(* IEC 61131-3 sources: Industry-PLC-LLM/data/PLCBEAD_repo/PLCBEAD_PLCEmbed-main/PLC-BEAD/Source/OpenPLCv2 (part 4) *)

(* ---- DIR_TO_DEG.ST ---- *)
TYPE oscat_LANGUAGE:
  STRUCT
    DEFAULT 	: INT;
	LMAX    	: INT;
  END_STRUCT;
END_TYPE

TYPE
  oscat_ELEMENT_DIRS 		: ARRAY [0..15] OF STRING;
  oscat_DIRS				: ARRAY [1..3]  OF oscat_ELEMENT_DIRS := [0,0 , 0];
END_TYPE

FUNCTION_BLOCK SETUP_DIRS
	VAR_IN_OUT
		DIRS :	oscat_DIRS;
	END_VAR

	VAR
		init :	BOOL;
	END_VAR

	IF init THEN RETURN; END_IF;
	init := TRUE;

	(* ---- english --- *)
	DIRS[1][00] := 'N';
	DIRS[1][01] := 'NNE';
	DIRS[1][02] := 'NE';
	DIRS[1][03] := 'ENE';
	DIRS[1][04] := 'E';
	DIRS[1][05] := 'ESE';
	DIRS[1][06] := 'SE';
	DIRS[1][07] := 'SSE';
	DIRS[1][08] := 'S';
	DIRS[1][09] := 'SSW';
	DIRS[1][10] := 'SW';
	DIRS[1][11] := 'WSW';
	DIRS[1][12] := 'W';
	DIRS[1][13] := 'WNW';
	DIRS[1][14] := 'NW';
	DIRS[1][15] := 'NNW';

	(* ---- german --- *)
	DIRS[2][00] := 'N';
	DIRS[2][01] := 'NNO';
	DIRS[2][02] := 'NO';
	DIRS[2][03] := 'ONO';
	DIRS[2][04] := 'O';
	DIRS[2][05] := 'OSO';
	DIRS[2][06] := 'SO';
	DIRS[2][07] := 'SSO';
	DIRS[2][08] := 'S';
	DIRS[2][09] := 'SSW';
	DIRS[2][10] := 'SW';
	DIRS[2][11] := 'WSW';
	DIRS[2][12] := 'W';
	DIRS[2][13] := 'WNW';
	DIRS[2][14] := 'NW';
	DIRS[2][15] := 'NNW';

	(* ---- french --- *)
	DIRS[3][00] := 'N';
	DIRS[3][01] := 'NNO';
	DIRS[3][02] := 'NO';
	DIRS[3][03] := 'ONO';
	DIRS[3][04] := 'O';
	DIRS[3][05] := 'OSO';
	DIRS[3][06] := 'SO';
	DIRS[3][07] := 'SSO';
	DIRS[3][08] := 'S';
	DIRS[3][09] := 'SSW';
	DIRS[3][10] := 'SW';
	DIRS[3][11] := 'WSW';
	DIRS[3][12] := 'W';
	DIRS[3][13] := 'WNW';
	DIRS[3][14] := 'NW';
	DIRS[3][15] := 'NNW';
END_FUNCTION_BLOCK

FUNCTION_BLOCK SETUP_LANGUAGE_Block

	VAR_IN_OUT
		LANGUAGE :	oscat_LANGUAGE;
	END_VAR

	VAR
		init :	BOOL;
	END_VAR

	IF init THEN RETURN; END_IF;
	init := TRUE;

	LANGUAGE.DEFAULT  := 1; (* 1=english, 2=german 3=french *)
	LANGUAGE.LMAX := 3;

END_FUNCTION_BLOCK

FUNCTION_BLOCK DIR_TO_DEG_Block
	VAR_INPUT
		DIR :	STRING;
		L :	INT;
	END_VAR

	VAR_OUTPUT
		DIR_TO_DEG :	INT;
	END_VAR

	VAR
		ly :	INT;
		i :	INT;
		SETUP_DIRSS :	SETUP_DIRS;
		DIRS :	oscat_DIRS;
		SETUP_LANGUAGE :	SETUP_LANGUAGE_Block;
		LANGUAGE :	oscat_LANGUAGE;
	END_VAR

	SETUP_DIRSS(DIRS:=DIRS);
	DIRS:=SETUP_DIRSS.DIRS;
	SETUP_LANGUAGE(LANGUAGE:=LANGUAGE);
	LANGUAGE:=SETUP_LANGUAGE.LANGUAGE;

	IF L = 0 THEN ly := LANGUAGE.DEFAULT; ELSE ly := MIN(L, LANGUAGE.LMAX); END_IF;
	FOR i := 0 TO 15 DO
		IF EQ_STRING(DIRS[ly][i],DIR) THEN EXIT; END_IF;
	END_FOR;
	DIR_TO_DEG := WORD_TO_INT(SHR(INT_TO_WORD(i * 45 + 1), 1));

END_FUNCTION_BLOCK

PROGRAM program0
  VAR
    LocalVar0 : STRING;
	LocalVar1 : INT;

	LocalOUT  : INT;
	func_block : DIR_TO_DEG_Block;
  END_VAR
	func_block.DIR  := LocalVar0;
	func_block.L  := LocalVar1;
	func_block();
	LocalOUT := func_block.DIR_TO_DEG;
END_PROGRAM

CONFIGURATION Config0
  RESOURCE Res0 ON PLC
    TASK task0(INTERVAL := T#20ms,PRIORITY := 0);
    PROGRAM instance0 WITH task0 : program0;
  END_RESOURCE
END_CONFIGURATION

(* ---- DRIVER_1.ST ---- *)
FUNCTION_BLOCK DRIVER_1
	VAR_INPUT
		SET :	BOOL;
		IN :	BOOL;
		RST :	BOOL;
		TOGGLE_MODE :	BOOL;
		TIMEOUT :	TIME;
	END_VAR

	VAR_OUTPUT
		Q :	BOOL;
	END_VAR

	VAR
		off :	TON;
		edge :	BOOL;
	END_VAR

	IF off.Q THEN Q := FALSE; END_IF;
	IF rst THEN
		Q := FALSE;
	ELSIF set THEN
		Q := TRUE;
	ELSIF IN AND NOT edge THEN
		IF toggle_mode THEN q := NOT Q; ELSE q := TRUE; END_IF;
	END_IF;
	edge := in;
	IF timeout > t#0s THEN off(in := Q, PT := Timeout); END_IF;

END_FUNCTION_BLOCK

PROGRAM program0
  VAR
	SET         :	BOOL;
	IN          :	BOOL;
	RST         :	BOOL;
	TOGGLE_MODE :	BOOL;
	TIMEOUT     :	TIME;

	Q :	BOOL;

	func_block : DRIVER_1;
  END_VAR
	func_block.SET         :=SET        ;
	func_block.IN          :=IN         ;
	func_block.RST         :=RST        ;
	func_block.TOGGLE_MODE :=TOGGLE_MODE;
	func_block.TIMEOUT     :=TIMEOUT    ;
	func_block();
	Q := func_block.Q;
END_PROGRAM

CONFIGURATION Config0
  RESOURCE Res0 ON PLC
    TASK task0(INTERVAL := T#20ms,PRIORITY := 0);
    PROGRAM instance0 WITH task0 : program0;
  END_RESOURCE
END_CONFIGURATION

(* ---- DRIVER_4.ST ---- *)
FUNCTION_BLOCK DRIVER_1
	VAR_INPUT
		SET :	BOOL;
		IN :	BOOL;
		RST :	BOOL;
		TOGGLE_MODE :	BOOL;
		TIMEOUT :	TIME;
	END_VAR

	VAR_OUTPUT
		Q :	BOOL;
	END_VAR

	VAR
		off :	TON;
		edge :	BOOL;
	END_VAR

	IF off.Q THEN Q := FALSE; END_IF;
	IF rst THEN
		Q := FALSE;
	ELSIF set THEN
		Q := TRUE;
	ELSIF IN AND NOT edge THEN
		IF toggle_mode THEN q := NOT Q; ELSE q := TRUE; END_IF;
	END_IF;
	edge := in;
	IF timeout > t#0s THEN off(in := Q, PT := Timeout); END_IF;

END_FUNCTION_BLOCK

FUNCTION_BLOCK DRIVER_4

	VAR_INPUT
		SET :	BOOL;
		IN0 :	BOOL;
		IN1 :	BOOL;
		IN2 :	BOOL;
		IN3 :	BOOL;
		RST :	BOOL;
		TOGGLE_MODE :	BOOL;
		TIMEOUT :	TIME;
	END_VAR

	VAR_OUTPUT
		Q0 :	BOOL;
		Q1 :	BOOL;
		Q2 :	BOOL;
		Q3 :	BOOL;
	END_VAR

	VAR
		d0 :	DRIVER_1;
		d1 :	DRIVER_1;
		d2 :	DRIVER_1;
		d3 :	DRIVER_1;
	END_VAR

	D0(Set:=set, in:=in0, rst:=rst, toggle_mode:=toggle_mode, timeout:=timeout);
	D1(Set:=set, in:=in1, rst:=rst, toggle_mode:=toggle_mode, timeout:=timeout);
	D2(Set:=set, in:=in2, rst:=rst, toggle_mode:=toggle_mode, timeout:=timeout);
	D3(Set:=set, in:=in3, rst:=rst, toggle_mode:=toggle_mode, timeout:=timeout);
	Q0 := D0.Q;
	Q1 := D1.Q;
	Q2 := D2.Q;
	Q3 := D3.Q;

END_FUNCTION_BLOCK

PROGRAM program0
  VAR
	SET         :	BOOL;
	IN0         :	BOOL;
	IN1         :	BOOL;
	IN2         :	BOOL;
	IN3         :	BOOL;
	RST         :	BOOL;
	TOGGLE_MODE :	BOOL;
	TIMEOUT     :	TIME;

	Q0 :	BOOL;
	Q1 :	BOOL;
	Q2 :	BOOL;
	Q3 :	BOOL;

	func_block : DRIVER_4;
  END_VAR
	func_block.SET         := SET        ;
	func_block.IN0         := IN0        ;
	func_block.IN1         := IN1        ;
	func_block.IN2         := IN2        ;
	func_block.IN3         := IN3        ;
	func_block.RST         := RST        ;
	func_block.TOGGLE_MODE := TOGGLE_MODE;
	func_block.TIMEOUT     := TIMEOUT    ;
	func_block();
	Q0 := func_block.Q0;
	Q1 := func_block.Q1;
	Q2 := func_block.Q2;
	Q3 := func_block.Q3;
END_PROGRAM

CONFIGURATION Config0
  RESOURCE Res0 ON PLC
    TASK task0(INTERVAL := T#20ms,PRIORITY := 0);
    PROGRAM instance0 WITH task0 : program0;
  END_RESOURCE
END_CONFIGURATION

(* ---- DRIVER_4C.ST ---- *)
TYPE
  oscat_DRIVER_4C 			  : ARRAY [1..7] 	OF BYTE;
END_TYPE
FUNCTION_BLOCK DRIVER_4C

	VAR_INPUT
		IN :	BOOL;
		RST :	BOOL;
		TIMEOUT :	TIME;
		SX :	oscat_DRIVER_4C;
	END_VAR

	VAR_OUTPUT
		SN :	INT;
		Q0 :	BOOL;
		Q1 :	BOOL;
		Q2 :	BOOL;
		Q3 :	BOOL;
	END_VAR

	VAR
		off :	TON;
		edge :	BOOL;
	END_VAR

	IF RST OR off.Q THEN
		SN := 0;
	ELSIF IN AND NOT edge THEN
		SN := SN + 1;
		IF SN > 7 OR SX[SN] = BYTE#0 THEN SN := 0; END_IF;
	END_IF;
	edge := in;
	IF SN > 0 THEN
		Q0 := (SX[SN] AND BYTE#1) > BYTE#0;
		Q1 := (SX[SN] AND BYTE#2) > BYTE#0;
		Q2 := (SX[SN] AND BYTE#4) > BYTE#0;
		Q3 := (SX[SN] AND BYTE#8) > BYTE#0;
	ELSE
		Q0 := FALSE;
		Q1 := FALSE;
		Q2 := FALSE;
		Q3 := FALSE;
	END_IF;

	IF timeout > t#0s THEN off(in := SN > 0, PT := Timeout); END_IF;

END_FUNCTION_BLOCK

PROGRAM program0
  VAR
	IN      :	BOOL;
	RST     :	BOOL;
	TIMEOUT :	TIME;
	SX      :	oscat_DRIVER_4C;

	SN :	INT;
	Q0 :	BOOL;
	Q1 :	BOOL;
	Q2 :	BOOL;
	Q3 :	BOOL;

	func_block : DRIVER_4C;
  END_VAR
	func_block.IN       :=IN      ;
	func_block.RST      :=RST     ;
	func_block.TIMEOUT  :=TIMEOUT ;
	func_block.SX       :=SX      ;
	func_block();
	SN := func_block.SN;
	Q0 := func_block.Q0;
	Q1 := func_block.Q1;
	Q2 := func_block.Q2;
	Q3 := func_block.Q3;
END_PROGRAM

CONFIGURATION Config0
  RESOURCE Res0 ON PLC
    TASK task0(INTERVAL := T#20ms,PRIORITY := 0);
    PROGRAM instance0 WITH task0 : program0;
  END_RESOURCE
END_CONFIGURATION

(* ---- DT2_TO_SDT.ST ---- *)
TYPE oscat_SDT :
STRUCT
	YEAR : INT;
	MONTH : INT;
	DAY : INT;
	WEEKDAY : INT;
	HOUR : INT;
	MINUTE : INT;
	SECOND : INT;
	MS : INT;
END_STRUCT;
END_TYPE

FUNCTION DAY_OF_WEEK:INT

	VAR_INPUT
		IDATE :	UDINT;
	END_VAR

	DAY_OF_WEEK := UDINT_TO_INT((idate / UDINT#86400 + UDINT#3) MOD UDINT#7) + INT#01;
END_FUNCTION

FUNCTION DAY_OF_YEAR:INT
	VAR_INPUT
		IDATE :	UDINT;
	END_VAR

	DAY_OF_YEAR := UDINT_TO_INT(((idate) / UDINT#86400) MOD UDINT#1461);
	IF DAY_OF_YEAR > 729 THEN
		IF DAY_OF_YEAR > 1095 THEN DAY_OF_YEAR := DAY_OF_YEAR - 1095; ELSE DAY_OF_YEAR := DAY_OF_YEAR - 729; END_IF;
	ELSIF DAY_OF_YEAR > 364 THEN
		DAY_OF_YEAR := DAY_OF_YEAR - 364;
	ELSE
		DAY_OF_YEAR := DAY_OF_YEAR + 1;
	END_IF;
END_FUNCTION

FUNCTION LEAP_OF_DATE:BOOL

	VAR_INPUT
		IDATE :	UDINT;
	END_VAR

	LEAP_OF_DATE := SHL(UDINT_TO_DWORD((idate + UDINT#43200) / UDINT#31557600), 30) = DWORD#16#80000000;
END_FUNCTION

FUNCTION DAY_OF_MONTH:INT
	VAR_INPUT
		IDATE :	UDINT;
	END_VAR

	day_of_month := day_of_year(idate);

	IF leap_of_Date(idate) THEN
		CASE day_of_month OF
			32..60	:	day_of_month := day_of_month - 31;
			61..91	:	day_of_month := day_of_month - 60;
			92..121 :	day_of_month := day_of_month - 91;
			122..152:	day_of_month := day_of_month - 121;
			153..182:	day_of_month := day_of_month - 152;
			183..213:	day_of_month := day_of_month - 182;
			214..244:	day_of_month := day_of_month - 213;
			245..274:	day_of_month := day_of_month - 244;
			275..305:	day_of_month := day_of_month - 274;
			306..335:	day_of_month := day_of_month - 305;
			336..366:	day_of_month := day_of_month - 335;
		END_CASE;
	ELSE
		CASE day_of_month OF
			32..59	:	day_of_month := day_of_month - 31;
			60..90	:	day_of_month := day_of_month - 59;
			91..120 :	day_of_month := day_of_month - 90;
			121..151:	day_of_month := day_of_month - 120;
			152..181:	day_of_month := day_of_month - 151;
			182..212:	day_of_month := day_of_month - 181;
			213..243:	day_of_month := day_of_month - 212;
			244..273:	day_of_month := day_of_month - 243;
			274..304:	day_of_month := day_of_month - 273;
			305..334:	day_of_month := day_of_month - 304;
			335..365:	day_of_month := day_of_month - 334;
		END_CASE;
	END_IF;
END_FUNCTION

FUNCTION MONTH_OF_DATE:INT

	VAR_INPUT
		IDATE :	UDINT;
	END_VAR

	MONTH_OF_DATE := DAY_OF_YEAR(idate);
	IF MONTH_OF_DATE < 32 THEN
		MONTH_OF_DATE := 1;
	ELSIF LEAP_OF_DATE((IDATE)) THEN
		MONTH_OF_DATE := (MONTH_OF_DATE * 53 + 1668) / 1623;
	ELSE
		MONTH_OF_DATE := (MONTH_OF_DATE * 53 + 1700) / 1620;
	END_IF;
END_FUNCTION

FUNCTION YEAR_OF_DATE:INT
	VAR_INPUT
		IDATE :	UDINT;
	END_VAR

	YEAR_OF_DATE := UDINT_TO_INT((idate+UDINT#43200) / UDINT#31557600 + UDINT#1970);
END_FUNCTION

FUNCTION_BLOCK DT2_TO_SDT
VAR_INPUT
	DI :	UDINT;
	TI :	UDINT;
END_VAR

VAR_OUTPUT
	SDT :	oscat_SDT;
END_VAR

SDT.YEAR := YEAR_OF_DATE(di);
SDT.MONTH := MONTH_OF_DATE(di);
SDT.DAY := DAY_OF_MONTH(di);
SDT.WEEKDAY := DAY_OF_WEEK(di);
SDT.MS := UDINT_TO_INT(ti MOD UDINT#1000);
SDT.SECOND := UDINT_TO_INT((ti / UDINT#1000) MOD UDINT#60);
SDT.MINUTE := UDINT_TO_INT((ti / UDINT#60000) MOD UDINT#60);
SDT.HOUR := UDINT_TO_INT(ti / UDINT#3600000);

END_FUNCTION_BLOCK

PROGRAM program0
  VAR
    LocalVar0 : UDINT;
	LocalVar1 : UDINT;
	LocalOUT  : oscat_SDT;
	func_block : DT2_TO_SDT;
  END_VAR
	func_block.DI  := LocalVar0;
	func_block.TI  := LocalVar1;
	func_block();
	LocalOUT := func_block.SDT;
END_PROGRAM

CONFIGURATION Config0
  RESOURCE Res0 ON PLC
    TASK task0(INTERVAL := T#20ms,PRIORITY := 0);
    PROGRAM instance0 WITH task0 : program0;
  END_RESOURCE
END_CONFIGURATION

(* ---- DT_SIMU.ST ---- *)
FUNCTION _REAL_TO_UDINT:UDINT
  VAR_INPUT
    X :	REAL;
  END_VAR

  IF REAL_TO_UDINT(0.5) = UDINT#1 THEN
    _REAL_TO_UDINT := REAL_TO_UDINT(x);
  ELSIF X > 0.0 THEN
    _REAL_TO_UDINT := REAL_TO_UDINT(x+0.5);
  ELSIF X < 0.0 THEN
    _REAL_TO_UDINT := REAL_TO_UDINT(x-0.5);
  ELSE
    _REAL_TO_UDINT := UDINT#0;
  END_IF;
END_FUNCTION

FUNCTION_BLOCK T_PLC_MS_block

	VAR_OUTPUT
		T_PLC_MS :	UDINT;
	END_VAR

	VAR_EXTERNAL
		PLC_TICKS_PER_SEC :	INT;
		PLC_SYS_TICK_CNT :	DINT;
	END_VAR

	VAR
		debug :	BOOL;(*Debug-Mode ON / OFF*)
		N :	INT;(*Debug-Faktor*)
		Offset :	UDINT;(*Debug-Offset*)
		temp :	DWORD := DWORD#1;(*Debug-Offset*)
		mode :	BOOL;(*modus*)
		faktor :	UDINT;(*Systemtakt-Faktor*)
		init :	BOOL;
		v_plc_ticks_per_sec :	UDINT;
		base :	UDINT := UDINT#1000;
	END_VAR

	IF init = FALSE THEN
		v_plc_ticks_per_sec := INT_TO_UDINT(PLC_TICKS_PER_SEC);
		IF v_plc_ticks_per_sec = UDINT#1024 THEN
			faktor := UDINT#1;
			mode := FALSE;
		ELSIF v_plc_ticks_per_sec > UDINT#0 THEN
			IF v_plc_ticks_per_sec <= base THEN
				faktor := base / v_plc_ticks_per_sec;
				mode := FALSE;
			ELSE
				faktor := v_plc_ticks_per_sec / base;
				mode := TRUE;
			END_IF;
		ELSE
			faktor := UDINT#1;
		END_IF;
		init := TRUE;
	END_IF;

	IF mode THEN
		T_PLC_MS := DINT_TO_UDINT(PLC_SYS_TICK_CNT) / faktor;
	ELSE
		T_PLC_MS := DINT_TO_UDINT(PLC_SYS_TICK_CNT) * faktor;
	END_IF;

	IF debug THEN
		T_PLC_MS := (DWORD_TO_UDINT(SHL(UDINT_TO_DWORD(T_PLC_MS),N) OR SHL(temp,N)) - UDINT#1) + Offset;
	END_IF;

END_FUNCTION_BLOCK

FUNCTION_BLOCK DT_SIMU
	VAR_INPUT
		START :	UDINT;
		SPEED :	REAL := 1.0;
	END_VAR

	VAR_OUTPUT
		DTS :	UDINT;
	END_VAR

	VAR
		tc :	UDINT;
		init :	BOOL;
		last :	UDINT;
		tx :	UDINT;
		td :	UDINT;
		T_PLC_MS :	T_PLC_MS_block;
	END_VAR

	T_PLC_MS();
	tx:= T_PLC_MS.T_PLC_MS;
	tc := _REAL_TO_UDINT(UDINT_TO_REAL(tx - last) * speed);

	IF NOT init THEN
		init := TRUE;
		DTS := Start;
		tc := UDINT#0;
		last := tx;
	ELSIF SPEED = 0.0 THEN
		DTS := DTS + UDINT#1;
	ELSIF tc >= UDINT#1000 THEN
		td := (tc / UDINT#1000) * UDINT#1000;
		DTS := DTS + td;
		last := last + _REAL_TO_UDINT(UDINT_TO_REAL(td) / speed);
	END_IF;
END_FUNCTION_BLOCK

PROGRAM program0
  VAR
    LocalVar0 : UDINT;
	LocalVar1 : REAL;
	LocalOUT  : UDINT;
	func_block : DT_SIMU;
  END_VAR
	func_block.START  := LocalVar0;
	func_block.SPEED  := LocalVar1;
	func_block();
	LocalOUT := func_block.DTS;
END_PROGRAM

CONFIGURATION Config0

	VAR_GLOBAL
		PLC_TICKS_PER_SEC :	INT;
		PLC_SYS_TICK_CNT :	DINT;
	END_VAR

  	RESOURCE Res0 ON PLC
    	TASK task0(INTERVAL := T#20ms,PRIORITY := 0);
    	PROGRAM instance0 WITH task0 : program0;
  	END_RESOURCE

END_CONFIGURATION

(* ---- DT_TO_SDT.ST ---- *)
TYPE oscat_SDT :
STRUCT
	YEAR : INT;
	MONTH : INT;
	DAY : INT;
	WEEKDAY : INT;
	HOUR : INT;
	MINUTE : INT;
	SECOND : INT;
	MS : INT;
END_STRUCT;
END_TYPE

FUNCTION DT_TO_DATE2:UDINT

	VAR_INPUT
		IN :	UDINT;
	END_VAR

	DT_TO_DATE2 := (IN / UDINT#86400) * UDINT#86400;
END_FUNCTION

FUNCTION YEAR_OF_DATE:INT
	VAR_INPUT
		IDATE :	UDINT;
	END_VAR

	YEAR_OF_DATE := UDINT_TO_INT((idate+UDINT#43200) / UDINT#31557600 + UDINT#1970);
END_FUNCTION

FUNCTION DAY_OF_WEEK:INT

	VAR_INPUT
		IDATE :	UDINT;
	END_VAR

	DAY_OF_WEEK := UDINT_TO_INT((idate / UDINT#86400 + UDINT#3) MOD UDINT#7) + INT#01;
END_FUNCTION

FUNCTION LEAP_OF_DATE:BOOL

	VAR_INPUT
		IDATE :	UDINT;
	END_VAR

	LEAP_OF_DATE := SHL(UDINT_TO_DWORD((idate + UDINT#43200) / UDINT#31557600), 30) = DWORD#16#80000000;
END_FUNCTION

FUNCTION DAY_OF_YEAR:INT
	VAR_INPUT
		IDATE :	UDINT;
	END_VAR

	DAY_OF_YEAR := UDINT_TO_INT(((idate) / UDINT#86400) MOD UDINT#1461);
	IF DAY_OF_YEAR > 729 THEN
		IF DAY_OF_YEAR > 1095 THEN DAY_OF_YEAR := DAY_OF_YEAR - 1095; ELSE DAY_OF_YEAR := DAY_OF_YEAR - 729; END_IF;
	ELSIF DAY_OF_YEAR > 364 THEN
		DAY_OF_YEAR := DAY_OF_YEAR - 364;
	ELSE
		DAY_OF_YEAR := DAY_OF_YEAR + 1;
	END_IF;
END_FUNCTION

FUNCTION MONTH_OF_DATE:INT

	VAR_INPUT
		IDATE :	UDINT;
	END_VAR

	MONTH_OF_DATE := DAY_OF_YEAR(idate);
	IF MONTH_OF_DATE < 32 THEN
		MONTH_OF_DATE := 1;
	ELSIF LEAP_OF_DATE((IDATE)) THEN
		MONTH_OF_DATE := (MONTH_OF_DATE * 53 + 1668) / 1623;
	ELSE
		MONTH_OF_DATE := (MONTH_OF_DATE * 53 + 1700) / 1620;
	END_IF;
END_FUNCTION

FUNCTION DAY_OF_MONTH:INT
	VAR_INPUT
		IDATE :	UDINT;
	END_VAR

	day_of_month := day_of_year(idate);

	IF leap_of_Date((idate)) THEN
		CASE day_of_month OF
			32..60	:	day_of_month := day_of_month - 31;
			61..91	:	day_of_month := day_of_month - 60;
			92..121 :	day_of_month := day_of_month - 91;
			122..152:	day_of_month := day_of_month - 121;
			153..182:	day_of_month := day_of_month - 152;
			183..213:	day_of_month := day_of_month - 182;
			214..244:	day_of_month := day_of_month - 213;
			245..274:	day_of_month := day_of_month - 244;
			275..305:	day_of_month := day_of_month - 274;
			306..335:	day_of_month := day_of_month - 305;
			336..366:	day_of_month := day_of_month - 335;
		END_CASE;
	ELSE
		CASE day_of_month OF
			32..59	:	day_of_month := day_of_month - 31;
			60..90	:	day_of_month := day_of_month - 59;
			91..120 :	day_of_month := day_of_month - 90;
			121..151:	day_of_month := day_of_month - 120;
			152..181:	day_of_month := day_of_month - 151;
			182..212:	day_of_month := day_of_month - 181;
			213..243:	day_of_month := day_of_month - 212;
			244..273:	day_of_month := day_of_month - 243;
			274..304:	day_of_month := day_of_month - 273;
			305..334:	day_of_month := day_of_month - 304;
			335..365:	day_of_month := day_of_month - 334;
		END_CASE;
	END_IF;
END_FUNCTION

FUNCTION _INT_TO_UDINT:UDINT
	VAR_INPUT
		IN :	INT;
	END_VAR

	_INT_TO_UDINT := DINT_TO_UDINT(INT_TO_DINT(IN));
END_FUNCTION

FUNCTION_BLOCK DT_TO_SDT

	VAR_INPUT
		DTI :	UDINT;
	END_VAR

	VAR_OUTPUT
		SDT :	oscat_SDT;
	END_VAR

	VAR
		tmp :	UDINT;
		tdt :	UDINT;
	END_VAR

	tmp := DT_TO_DATE2(dti);
	tdt := dti - tmp;
	SDT.YEAR := YEAR_OF_DATE(tmp);
	SDT.MONTH := MONTH_OF_DATE(tmp);
	SDT.DAY := DAY_OF_MONTH(tmp);
	SDT.WEEKDAY := DAY_OF_WEEK(tmp);
	SDT.SECOND := UDINT_TO_INT(tdt MOD UDINT#60);
	SDT.MINUTE := UDINT_TO_INT((tdt / UDINT#60) MOD UDINT#60);
	SDT.HOUR := UDINT_TO_INT(tdt / UDINT#3600);

END_FUNCTION_BLOCK

PROGRAM program0
  VAR
    LocalVar0 : UDINT;
	LocalOUT  : oscat_SDT;
	func_block : DT_TO_SDT;
  END_VAR
	func_block.DTI  := LocalVar0;
	func_block();
	LocalOUT := func_block.SDT;
END_PROGRAM

CONFIGURATION Config0
  RESOURCE Res0 ON PLC
    TASK task0(INTERVAL := T#20ms,PRIORITY := 0);
    PROGRAM instance0 WITH task0 : program0;
  END_RESOURCE
END_CONFIGURATION

(* ---- DT_TO_STRING.ST ---- *)
FUNCTION YEAR_OF_DATE:INT
	VAR_INPUT
		IDATE :	UDINT;
	END_VAR

	YEAR_OF_DATE := UDINT_TO_INT((idate+UDINT#43200) / UDINT#31557600 + UDINT#1970);
END_FUNCTION

FUNCTION DAY_OF_YEAR:INT
	VAR_INPUT
		IDATE :	UDINT;
	END_VAR

	DAY_OF_YEAR := UDINT_TO_INT(((idate) / UDINT#86400) MOD UDINT#1461);
	IF DAY_OF_YEAR > 729 THEN
		IF DAY_OF_YEAR > 1095 THEN DAY_OF_YEAR := DAY_OF_YEAR - 1095; ELSE DAY_OF_YEAR := DAY_OF_YEAR - 729; END_IF;
	ELSIF DAY_OF_YEAR > 364 THEN
		DAY_OF_YEAR := DAY_OF_YEAR - 364;
	ELSE
		DAY_OF_YEAR := DAY_OF_YEAR + 1;
	END_IF;
END_FUNCTION

FUNCTION LEAP_OF_DATE:BOOL

	VAR_INPUT
		IDATE :	UDINT;
	END_VAR

	LEAP_OF_DATE := SHL(UDINT_TO_DWORD((idate + UDINT#43200) / UDINT#31557600), 30) = DWORD#16#80000000;
END_FUNCTION

FUNCTION MONTH_OF_DATE:INT

	VAR_INPUT
		IDATE :	UDINT;
	END_VAR

	MONTH_OF_DATE := DAY_OF_YEAR(idate);
	IF MONTH_OF_DATE < 32 THEN
		MONTH_OF_DATE := 1;
	ELSIF LEAP_OF_DATE(IDATE) THEN
		MONTH_OF_DATE := (MONTH_OF_DATE * 53 + 1668) / 1623;
	ELSE
		MONTH_OF_DATE := (MONTH_OF_DATE * 53 + 1700) / 1620;
	END_IF;
END_FUNCTION

FUNCTION DAY_OF_MONTH:INT
	VAR_INPUT
		IDATE :	UDINT;
	END_VAR

	day_of_month := day_of_year(idate);

	IF leap_of_Date((idate)) THEN
		CASE day_of_month OF
			32..60	:	day_of_month := day_of_month - 31;
			61..91	:	day_of_month := day_of_month - 60;
			92..121 :	day_of_month := day_of_month - 91;
			122..152:	day_of_month := day_of_month - 121;
			153..182:	day_of_month := day_of_month - 152;
			183..213:	day_of_month := day_of_month - 182;
			214..244:	day_of_month := day_of_month - 213;
			245..274:	day_of_month := day_of_month - 244;
			275..305:	day_of_month := day_of_month - 274;
			306..335:	day_of_month := day_of_month - 305;
			336..366:	day_of_month := day_of_month - 335;
		END_CASE;
	ELSE
		CASE day_of_month OF
			32..59	:	day_of_month := day_of_month - 31;
			60..90	:	day_of_month := day_of_month - 59;
			91..120 :	day_of_month := day_of_month - 90;
			121..151:	day_of_month := day_of_month - 120;
			152..181:	day_of_month := day_of_month - 151;
			182..212:	day_of_month := day_of_month - 181;
			213..243:	day_of_month := day_of_month - 212;
			244..273:	day_of_month := day_of_month - 243;
			274..304:	day_of_month := day_of_month - 273;
			305..334:	day_of_month := day_of_month - 304;
			335..365:	day_of_month := day_of_month - 334;
		END_CASE;
	END_IF;
END_FUNCTION

FUNCTION SECOND_OF_DT:INT

	VAR_INPUT
		XDT :	UDINT;
	END_VAR

	SECOND_OF_DT := UDINT_TO_INT(XDT MOD UDINT#60);
END_FUNCTION

FUNCTION HOUR_OF_DT:INT
	VAR_INPUT
		XDT :	UDINT;
	END_VAR

	HOUR_OF_DT := UDINT_TO_INT((XDT MOD UDINT#86400) / UDINT#3600);
END_FUNCTION

FUNCTION MINUTE_OF_DT:INT
	VAR_INPUT
		XDT :	UDINT;
	END_VAR

	MINUTE_OF_DT := UDINT_TO_INT((XDT MOD UDINT#3600) / UDINT#60);
END_FUNCTION

FUNCTION_BLOCK DT_TO_STRING_Block

	VAR_INPUT
		IDT :	UDINT;
	END_VAR

	VAR_OUTPUT
		DT_STRING :	STRING;
	END_VAR

	VAR
		st_tmp1 :	STRING;
		st_tmp2 :	STRING;
	END_VAR

	st_tmp2 := CONCAT(INT_TO_STRING(YEAR_OF_DATE(IDT)),INT_TO_STRING(MONTH_OF_DATE(IDT)));
	st_tmp1 := CONCAT(INT_TO_STRING(day_of_month(IDT)),INT_TO_STRING(hour_of_DT(IDT)));
	st_tmp2 := CONCAT(st_tmp2,st_tmp1);
	st_tmp1 := CONCAT(INT_TO_STRING(minute_of_DT(IDT)),INT_TO_STRING(second_of_DT(IDT)));
	st_tmp2 := CONCAT(st_tmp2,st_tmp1);
	DT_STRING := st_tmp2;
END_FUNCTION_BLOCK

PROGRAM program0
	VAR
		IDT : UDINT;
		OUT  : STRING;
		func_block : DT_TO_STRING_Block;
	END_VAR
	func_block.IDT := IDT;
	func_block();
	OUT := func_block.DT_STRING;
END_PROGRAM

CONFIGURATION Config0
	RESOURCE Res0 ON PLC
		TASK task0(INTERVAL := T#20ms,PRIORITY := 0);
		PROGRAM instance0 WITH task0 : program0;
	END_RESOURCE
END_CONFIGURATION

(* ---- DWORD_TO_STRB.ST ---- *)
FUNCTION_BLOCK DWORD_TO_STRB_Block
	VAR_INPUT
		IN :	DWORD;
	END_VAR

	VAR_OUTPUT
		DWORD_TO_STRB :	STRING;
	END_VAR

	VAR
		i :	INT;
	END_VAR

	DWORD_TO_STRB :='';
	FOR i := 1 TO 32 DO
		IF (in AND DWORD#16#8000_0000) > DWORD#0 THEN
			DWORD_TO_STRB := CONCAT(DWORD_TO_STRB,'1');
		ELSE
			DWORD_TO_STRB := CONCAT(DWORD_TO_STRB,'0');
		END_IF;
		in := SHL(in, 1);
	END_FOR;
END_FUNCTION_BLOCK

PROGRAM program0
  VAR
    IN :	DWORD;

	DWORD_TO_STRB :	STRING;
	func_block : DWORD_TO_STRB_Block;
  END_VAR
	func_block.IN  := IN;
	func_block();
	DWORD_TO_STRB := func_block.DWORD_TO_STRB;
END_PROGRAM

CONFIGURATION Config0
  RESOURCE Res0 ON PLC
    TASK task0(INTERVAL := T#20ms,PRIORITY := 0);
    PROGRAM instance0 WITH task0 : program0;
  END_RESOURCE
END_CONFIGURATION

(* ---- DWORD_TO_STRF.ST ---- *)
FUNCTION_BLOCK DWORD_TO_STRF_Block

	VAR_INPUT
		IN :	DWORD;
		N :	INT;
	END_VAR

	VAR_OUTPUT
		DWORD_TO_STRF :	STRING;
	END_VAR

	VAR
		temp :	STRING;
		temp2 :	STRING;
		L : INT;
	END_VAR

	temp := DWORD_TO_STRING(in);
	L := LEN(temp);
	IF N < L THEN
		temp :=RIGHT(temp,N);
		L := N;
	END_IF;

	WHILE L < N DO
		temp2 := temp;
		temp := CONCAT('0', temp2);
		L := L + 1;
	END_WHILE;
	DWORD_TO_STRF := temp;

END_FUNCTION_BLOCK

PROGRAM program0
  VAR
    IN :	DWORD;
	N :		INT;
	DWORD_TO_STRF :	STRING;
	func_block : DWORD_TO_STRF_Block;
  END_VAR
	func_block.IN  := IN;
	func_block.N  := N;
	func_block();
	DWORD_TO_STRF := func_block.DWORD_TO_STRF;
END_PROGRAM

CONFIGURATION Config0
  RESOURCE Res0 ON PLC
    TASK task0(INTERVAL := T#20ms,PRIORITY := 0);
    PROGRAM instance0 WITH task0 : program0;
  END_RESOURCE
END_CONFIGURATION

(* ---- DWORD_TO_STRH.ST ---- *)
FUNCTION_BLOCK DWORD_TO_STRH_Block

	VAR_INPUT
		IN :	DWORD;
	END_VAR

	VAR_OUTPUT
		DWORD_TO_STRH :	STRING;
	END_VAR

	DWORD_TO_STRH:=DWORD_TO_STRING(IN);

END_FUNCTION_BLOCK

PROGRAM program0
  VAR
    LocalVar0 : DWORD;
	LocalOUT  : STRING;
	func_block : DWORD_TO_STRH_Block;
  END_VAR
	func_block.IN  := LocalVar0;
	func_block();
	LocalOUT := func_block.DWORD_TO_STRH;
END_PROGRAM

CONFIGURATION Config0
  RESOURCE Res0 ON PLC
    TASK task0(INTERVAL := T#20ms,PRIORITY := 0);
    PROGRAM instance0 WITH task0 : program0;
  END_RESOURCE
END_CONFIGURATION

(* ---- ENERGY.ST ---- *)
FUNCTION_BLOCK ENERGY
	VAR_INPUT
		J :	REAL;
		C :	REAL;
		WH :	REAL;
	END_VAR

	VAR_OUTPUT
		YJ :	REAL;
		YC :	REAL;
		YWH :	REAL;
	END_VAR

	YJ := J + Wh * 3600.0 + C * 4.1868;
	YC := YJ * 0.238845896627496;
	YWh := YJ * 2.7777777778E-004;
END_FUNCTION_BLOCK

PROGRAM program0
  VAR
		J  :	REAL;
		C  :	REAL;
		WH :	REAL;

		YJ  :	REAL;
		YC  :	REAL;
		YWH :	REAL;
	func_block : ENERGY;
  END_VAR
	func_block.J  :=J ;
	func_block.C  :=C ;
	func_block.WH :=WH;
	func_block();
	YJ  := func_block.YJ ;
	YC  := func_block.YC ;
	YWH := func_block.YWH;

END_PROGRAM

CONFIGURATION Config0
	RESOURCE Res0 ON PLC
		TASK task0(INTERVAL := T#20ms,PRIORITY := 0);
		PROGRAM instance0 WITH task0 : program0;
	END_RESOURCE
END_CONFIGURATION

(* ---- ESR_COLLECT.ST ---- *)
TYPE
	oscat_esr_collect_data      : ARRAY [0..7]    OF BYTE;
END_TYPE
TYPE oscat_esr_data :
  STRUCT
	typ    : BYTE;
	adress : STRING;
	DS     : UDINT;
	TS     : TIME;
	data   : oscat_esr_collect_data;
  END_STRUCT;
END_TYPE

TYPE
  oscat_ESR_3                : ARRAY [0..3] OF oscat_esr_data;
  oscat_ESR_31               : ARRAY [0..31] OF oscat_esr_data;
END_TYPE

FUNCTION INC1:INT

	VAR_INPUT
		X :	INT;
		N :	INT;
	END_VAR

	IF X >= N - 1 THEN
		INC1 := 0;
	ELSE
		INC1 := X + 1;
	END_IF;
END_FUNCTION

FUNCTION_BLOCK ESR_COLLECT
	VAR_INPUT
		ESR_0 :	oscat_ESR_3;
		ESR_1 :	oscat_ESR_3;
		ESR_2 :	oscat_ESR_3;
		ESR_3 :	oscat_ESR_3;
		ESR_4 :	oscat_ESR_3;
		ESR_5 :	oscat_ESR_3;
		ESR_6 :	oscat_ESR_3;
		ESR_7 :	oscat_ESR_3;
		RST :	BOOL;
	END_VAR

	VAR_IN_OUT
		POS :	INT;
	END_VAR

	VAR_OUTPUT
		ESR_OUT :	oscat_ESR_31;
	END_VAR

	VAR
		cnt :	INT := -1;
		max_in :	INT := 3;
		max_out :	INT := 32;
	END_VAR

	IF rst OR cnt < 0 THEN
		pos := -1;
	ELSE
		FOR cnt := 0 TO max_in DO
		IF esr_0[cnt].typ > BYTE#0 THEN pos := INC1(pos, max_out); esr_out[pos] := esr_0[cnt]; END_IF;
		IF esr_1[cnt].typ > BYTE#0 THEN pos := INC1(pos, max_out); esr_out[pos] := esr_1[cnt]; END_IF;
		IF esr_2[cnt].typ > BYTE#0 THEN pos := INC1(pos, max_out); esr_out[pos] := esr_2[cnt]; END_IF;
		IF esr_3[cnt].typ > BYTE#0 THEN pos := INC1(pos, max_out); esr_out[pos] := esr_3[cnt]; END_IF;
		IF esr_4[cnt].typ > BYTE#0 THEN pos := INC1(pos, max_out); esr_out[pos] := esr_4[cnt]; END_IF;
		IF esr_5[cnt].typ > BYTE#0 THEN pos := INC1(pos, max_out); esr_out[pos] := esr_5[cnt]; END_IF;
		IF esr_6[cnt].typ > BYTE#0 THEN pos := INC1(pos, max_out); esr_out[pos] := esr_6[cnt]; END_IF;
		IF esr_7[cnt].typ > BYTE#0 THEN pos := INC1(pos, max_out); esr_out[pos] := esr_7[cnt]; END_IF;
	END_FOR;
	END_IF;

END_FUNCTION_BLOCK

PROGRAM program0
  VAR
	ESR_0 :	oscat_ESR_3;
	ESR_1 :	oscat_ESR_3;
	ESR_2 :	oscat_ESR_3;
	ESR_3 :	oscat_ESR_3;
	ESR_4 :	oscat_ESR_3;
	ESR_5 :	oscat_ESR_3;
	ESR_6 :	oscat_ESR_3;
	ESR_7 :	oscat_ESR_3;
	RST   :	BOOL;

	POS   :	INT;

	ESR_OUT :	oscat_ESR_31;

	func_block : ESR_COLLECT;
  END_VAR
	func_block.ESR_0 :=ESR_0;
	func_block.ESR_1 :=ESR_1;
	func_block.ESR_2 :=ESR_2;
	func_block.ESR_3 :=ESR_3;
	func_block.ESR_4 :=ESR_4;
	func_block.ESR_5 :=ESR_5;
	func_block.ESR_6 :=ESR_6;
	func_block.ESR_7 :=ESR_7;
	func_block.RST   :=RST  ;
	func_block.POS   :=POS  ;

	func_block();
	POS := func_block.POS;
	ESR_OUT := func_block.ESR_OUT;

END_PROGRAM

CONFIGURATION Config0
	RESOURCE Res0 ON PLC
		TASK task0(INTERVAL := T#20ms,PRIORITY := 0);
		PROGRAM instance0 WITH task0 : program0;
	END_RESOURCE
END_CONFIGURATION

(* ---- ESR_MON_B8.ST ---- *)
TYPE
	oscat_esr_collect_data      : ARRAY [0..7]    OF BYTE;
END_TYPE
TYPE oscat_esr_data :
  STRUCT
	typ    : BYTE;
	adress : STRING;
	DS     : UDINT;
	TS     : TIME;
	data   : oscat_esr_collect_data;
  END_STRUCT;
END_TYPE

TYPE
  oscat_ESR_3                : ARRAY [0..3] OF oscat_esr_data;
  oscat_ESR_31               : ARRAY [0..31] OF oscat_esr_data;
END_TYPE

FUNCTION_BLOCK T_PLC_MS_block

	VAR_OUTPUT
		T_PLC_MS :	UDINT;
	END_VAR

	VAR_EXTERNAL
		PLC_TICKS_PER_SEC :	INT;
		PLC_SYS_TICK_CNT :	DINT;
	END_VAR

	VAR
		debug :	BOOL;(*Debug-Mode ON / OFF*)
		N :	INT;(*Debug-Faktor*)
		Offset :	UDINT;(*Debug-Offset*)
		temp :	DWORD := DWORD#1;(*Debug-Offset*)
		mode :	BOOL;(*modus*)
		faktor :	UDINT;(*Systemtakt-Faktor*)
		init :	BOOL;
		v_plc_ticks_per_sec :	UDINT;
		base :	UDINT := UDINT#1000;
	END_VAR

	IF init = FALSE THEN
		v_plc_ticks_per_sec := INT_TO_UDINT(PLC_TICKS_PER_SEC);
		IF v_plc_ticks_per_sec = UDINT#1024 THEN
			faktor := UDINT#1;
			mode := FALSE;
		ELSIF v_plc_ticks_per_sec > UDINT#0 THEN
			IF v_plc_ticks_per_sec <= base THEN
				faktor := base / v_plc_ticks_per_sec;
				mode := FALSE;
			ELSE
				faktor := v_plc_ticks_per_sec / base;
				mode := TRUE;
			END_IF;
		ELSE
			faktor := UDINT#1;
		END_IF;
		init := TRUE;
	END_IF;

	IF mode THEN
		T_PLC_MS := DINT_TO_UDINT(PLC_SYS_TICK_CNT) / faktor;
	ELSE
		T_PLC_MS := DINT_TO_UDINT(PLC_SYS_TICK_CNT) * faktor;
	END_IF;

	IF debug THEN
		T_PLC_MS := (DWORD_TO_UDINT(SHL(UDINT_TO_DWORD(T_PLC_MS),N) OR SHL(temp,N)) - UDINT#1) + Offset;
	END_IF;

END_FUNCTION_BLOCK

FUNCTION_BLOCK ESR_MON_B8

	VAR_INPUT
		S0 :	BOOL;
		A0 :	STRING;
		S1 :	BOOL;
		A1 :	STRING;
		S2 :	BOOL;
		A2 :	STRING;
		S3 :	BOOL;
		A3 :	STRING;
		S4 :	BOOL;
		A4 :	STRING;
		S5 :	BOOL;
		A5 :	STRING;
		S6 :	BOOL;
		A6 :	STRING;
		S7 :	BOOL;
		A7 :	STRING;
		DT_IN :	UDINT;
	END_VAR

	VAR_IN_OUT
		ESR_Out :	oscat_ESR_3;
	END_VAR

	VAR_OUTPUT
		ESR_FLAG :	BOOL;
	END_VAR

	VAR
		x0 :	BOOL;
		x1 :	BOOL;
		x2 :	BOOL;
		x3 :	BOOL;
		x4 :	BOOL;
		x5 :	BOOL;
		x6 :	BOOL;
		x7 :	BOOL;
		tx :	TIME;
		cnt :	INT;
		T_PLC_MS :	T_PLC_MS_block;
	END_VAR

	T_PLC_MS();
	tx:= UDINT_TO_TIME(T_PLC_MS.T_PLC_MS);

	ESR_Flag := FALSE;
	esr_out[3].typ := BYTE#0;
	esr_out[2].typ := BYTE#0;
	esr_out[1].typ := BYTE#0;
	esr_out[0].typ := BYTE#0;
	cnt := 0;

	IF s0 <> X0 THEN
		esr_out[cnt].typ := INT_TO_BYTE(10 + BOOL_TO_INT(s0));
		esr_out[cnt].adress := a0;
		esr_out[cnt].DS := DT_in;
		esr_out[cnt].TS := TX;
		X0 := S0;
		cnt := cnt + 1;
		esr_flag := TRUE;
	END_IF;
	IF s1 <> X1 THEN
		esr_out[cnt].typ := INT_TO_BYTE(10 + BOOL_TO_INT(s1));
		esr_out[cnt].adress := a1;
		esr_out[cnt].DS := DT_in;
		esr_out[cnt].TS := TX;
		X1 := S1;
		cnt := cnt + 1;
		esr_flag := TRUE;
	END_IF;
	IF s2 <> X2 THEN
		esr_out[cnt].typ := INT_TO_BYTE(10 + BOOL_TO_INT(s2));
		esr_out[cnt].adress := a2;
		esr_out[cnt].DS := DT_in;
		esr_out[cnt].TS := TX;
		X2 := S2;
		cnt := cnt + 1;
		esr_flag := TRUE;
	END_IF;
	IF s3 <> X3 THEN
		esr_out[cnt].typ := INT_TO_BYTE(10 + BOOL_TO_INT(s3));
		esr_out[cnt].adress := a3;
		esr_out[cnt].DS := DT_in;
		esr_out[cnt].TS := TX;
		X3 := S3;
		cnt := cnt + 1;
		esr_flag := TRUE;
	END_IF;
	IF s4 <> X4 AND cnt < 4 THEN
		esr_out[cnt].typ := INT_TO_BYTE(10 + BOOL_TO_INT(s4));
		esr_out[cnt].adress := a4;
		esr_out[cnt].DS := DT_in;
		esr_out[cnt].TS := TX;
		X4 := S4;
		cnt := cnt + 1;
		esr_flag := TRUE;
	END_IF;
	IF s5 <> X5  AND cnt < 4 THEN
		esr_out[cnt].typ := INT_TO_BYTE(10 + BOOL_TO_INT(s5));
		esr_out[cnt].adress := a5;
		esr_out[cnt].DS := DT_in;
		esr_out[cnt].TS := TX;
		X5 := S5;
		cnt := cnt + 1;
		esr_flag := TRUE;
	END_IF;
	IF s6 <> X6  AND cnt < 4 THEN
		esr_out[cnt].typ := INT_TO_BYTE(10 + BOOL_TO_INT(s6));
		esr_out[cnt].adress := a6;
		esr_out[cnt].DS := DT_in;
		esr_out[cnt].TS := TX;
		X6 := S6;
		cnt := cnt + 1;
		esr_flag := TRUE;
	END_IF;
	IF s7 <> X7  AND cnt < 4 THEN
		esr_out[cnt].typ := INT_TO_BYTE(10 + BOOL_TO_INT(s7));
		esr_out[cnt].adress := a7;
		esr_out[cnt].DS := DT_in;
		esr_out[cnt].TS := TX;
		X7 := S7;
		cnt := cnt + 1;
		esr_flag := TRUE;
	END_IF;

END_FUNCTION_BLOCK

PROGRAM program0

	VAR

		S0 :	BOOL;
		A0 :	STRING;
		S1 :	BOOL;
		A1 :	STRING;
		S2 :	BOOL;
		A2 :	STRING;
		S3 :	BOOL;
		A3 :	STRING;
		S4 :	BOOL;
		A4 :	STRING;
		S5 :	BOOL;
		A5 :	STRING;
		S6 :	BOOL;
		A6 :	STRING;
		S7 :	BOOL;
		A7 :	STRING;
		DT_IN   :	UDINT;

		ESR_Out :	oscat_ESR_3;

		ESR_FLAG :	BOOL;

		func_block : ESR_MON_B8;
  	END_VAR
	func_block.S0 := S0;
	func_block.A0 := A0;
	func_block.S1 := S1;
	func_block.A1 := A1;
	func_block.S2 := S2;
	func_block.A2 := A2;
	func_block.S3 := S3;
	func_block.A3 := A3;
	func_block.S4 := S4;
	func_block.A4 := A4;
	func_block.S5 := S5;
	func_block.A5 := A5;
	func_block.S6 := S6;
	func_block.A6 := A6;
	func_block.S7 := S7;
	func_block.A7 := A7;
	func_block.DT_IN := DT_IN;
	func_block.ESR_Out := ESR_Out;
	func_block();
	ESR_Out := func_block.ESR_Out;
	ESR_FLAG := func_block.ESR_FLAG;

END_PROGRAM

CONFIGURATION Config0

	VAR_GLOBAL
		PLC_TICKS_PER_SEC :	INT;
		PLC_SYS_TICK_CNT :	DINT;
	END_VAR

  	RESOURCE Res0 ON PLC
    	TASK task0(INTERVAL := T#20ms,PRIORITY := 0);
    	PROGRAM instance0 WITH task0 : program0;
  	END_RESOURCE

END_CONFIGURATION

(* ---- ESR_MON_X8.ST ---- *)
TYPE
	oscat_esr_collect_data      : ARRAY [0..7]    OF BYTE;
END_TYPE

TYPE oscat_esr_data :
  STRUCT
	typ    : BYTE;
	adress : STRING;
	DS     : UDINT;
	TS     : TIME;
	data   : oscat_esr_collect_data;
  END_STRUCT;
END_TYPE

TYPE
  oscat_ESR_3                : ARRAY [0..3] OF oscat_esr_data;
  oscat_ESR_31               : ARRAY [0..31] OF oscat_esr_data;
END_TYPE

FUNCTION_BLOCK STATUS_TO_ESR_Block

	VAR_INPUT
		STATUS :	BYTE;
		ADRESS :	STRING;
		DT_IN :	UDINT;
		TS :	TIME;
	END_VAR

	VAR_OUTPUT
		STATUS_TO_ESR :	oscat_esr_data;
	END_VAR

	IF status < BYTE#100 THEN
		status_to_ESR.typ := BYTE#1;
	ELSIF status < BYTE#200 THEN
		status_to_ESR.typ := BYTE#2;
	ELSE
		status_to_ESR.typ := BYTE#3;
	END_IF;
	status_to_ESR.adress:= adress;
	status_to_ESR.DS := DT_in;
	status_to_ESR.TS := TS;
	status_to_ESR.data[0] := status;
END_FUNCTION_BLOCK

FUNCTION_BLOCK T_PLC_MS_block

	VAR_OUTPUT
		T_PLC_MS :	UDINT;
	END_VAR

	VAR_EXTERNAL
		PLC_TICKS_PER_SEC :	INT;
		PLC_SYS_TICK_CNT :	DINT;
	END_VAR

	VAR
		debug :	BOOL;(*Debug-Mode ON / OFF*)
		N :	INT;(*Debug-Faktor*)
		Offset :	UDINT;(*Debug-Offset*)
		temp :	DWORD := DWORD#1;(*Debug-Offset*)
		mode :	BOOL;(*modus*)
		faktor :	UDINT;(*Systemtakt-Faktor*)
		init :	BOOL;
		v_plc_ticks_per_sec :	UDINT;
		base :	UDINT := UDINT#1000;
	END_VAR

	IF init = FALSE THEN
		v_plc_ticks_per_sec := INT_TO_UDINT(PLC_TICKS_PER_SEC);
		IF v_plc_ticks_per_sec = UDINT#1024 THEN
			faktor := UDINT#1;
			mode := FALSE;
		ELSIF v_plc_ticks_per_sec > UDINT#0 THEN
			IF v_plc_ticks_per_sec <= base THEN
				faktor := base / v_plc_ticks_per_sec;
				mode := FALSE;
			ELSE
				faktor := v_plc_ticks_per_sec / base;
				mode := TRUE;
			END_IF;
		ELSE
			faktor := UDINT#1;
		END_IF;
		init := TRUE;
	END_IF;

	IF mode THEN
		T_PLC_MS := DINT_TO_UDINT(PLC_SYS_TICK_CNT) / faktor;
	ELSE
		T_PLC_MS := DINT_TO_UDINT(PLC_SYS_TICK_CNT) * faktor;
	END_IF;

	IF debug THEN
		T_PLC_MS := (DWORD_TO_UDINT(SHL(UDINT_TO_DWORD(T_PLC_MS),N) OR SHL(temp,N)) - UDINT#1) + Offset;
	END_IF;

END_FUNCTION_BLOCK

FUNCTION_BLOCK ESR_MON_X8
	VAR_INPUT
		S0 :	BYTE;
		A0 :	STRING;
		S1 :	BYTE;
		A1 :	STRING;
		S2 :	BYTE;
		A2 :	STRING;
		S3 :	BYTE;
		A3 :	STRING;
		S4 :	BYTE;
		A4 :	STRING;
		S5 :	BYTE;
		A5 :	STRING;
		S6 :	BYTE;
		A6 :	STRING;
		S7 :	BYTE;
		A7 :	STRING;
		DT_IN :	UDINT;
		MODE :	BYTE := BYTE#3;
	END_VAR

	VAR_IN_OUT
		ESR_OUT :	oscat_ESR_3;
	END_VAR

	VAR_OUTPUT
		ESR_FLAG :	BOOL;
	END_VAR

	VAR
		x0 :	BYTE;
		x1 :	BYTE;
		x2 :	BYTE;
		x3 :	BYTE;
		x4 :	BYTE;
		x5 :	BYTE;
		x6 :	BYTE;
		x7 :	BYTE;
		tx :	TIME;
		cnt :	INT;
		status_to_ESR :	STATUS_TO_ESR_Block;
		T_PLC_MS :	T_PLC_MS_block;
	END_VAR

	T_PLC_MS();
	tx:= UDINT_TO_TIME(T_PLC_MS.T_PLC_MS);

	ESR_Flag := FALSE;
	esr_out[3].typ := BYTE#0;
	esr_out[2].typ := BYTE#0;
	esr_out[1].typ := BYTE#0;
	esr_out[0].typ := BYTE#0;
	cnt := 0;

	IF s0 <> X0 AND ((s0 < BYTE#100) OR (S0 > BYTE#99 AND S0 < BYTE#200 AND mode >= BYTE#2) OR (S0 > BYTE#199 AND mode = BYTE#3)) THEN

		status_to_ESR.status := s0;
		status_to_ESR.adress := a0;
		status_to_ESR.DT_in  := DT_in;
		status_to_ESR.TS     := tx;
		status_to_ESR();
		esr_out[cnt] := status_to_ESR.status_to_ESR;

		X0 := S0;
		cnt := cnt + 1;
		esr_flag := TRUE;
	END_IF;
	IF s1 <> X1 AND ((s1 < BYTE#100) OR (S1 > BYTE#99 AND S1 < BYTE#200 AND mode >= BYTE#2) OR (S1 > BYTE#199 AND mode = BYTE#3)) THEN

		status_to_ESR.status := s1;
		status_to_ESR.adress := a1;
		status_to_ESR.DT_in  := DT_in;
		status_to_ESR.TS     := tx;
		status_to_ESR();
		esr_out[cnt] := status_to_ESR.status_to_ESR;

		X1 := S1;
		cnt := cnt + 1;
		esr_flag := TRUE;
	END_IF;
	IF s2 <> X2 AND ((s2 < BYTE#100) OR (S2 > BYTE#99 AND S2 < BYTE#200 AND mode >= BYTE#2) OR (S2 > BYTE#199 AND mode = BYTE#3)) THEN

		status_to_ESR.status := s2;
		status_to_ESR.adress := a2;
		status_to_ESR.DT_in  := DT_in;
		status_to_ESR.TS     := tx;
		status_to_ESR();
		esr_out[cnt] := status_to_ESR.status_to_ESR;

		X2 := S2;
		cnt := cnt + 1;
		esr_flag := TRUE;
	END_IF;
	IF s3 <> X3 AND ((s3 < BYTE#100) OR (S3 > BYTE#99 AND S3 < BYTE#200 AND mode >= BYTE#2) OR (S3 > BYTE#199 AND mode = BYTE#3)) THEN

		status_to_ESR.status := s3;
		status_to_ESR.adress := a3;
		status_to_ESR.DT_in  := DT_in;
		status_to_ESR.TS     := tx;
		status_to_ESR();
		esr_out[cnt] := status_to_ESR.status_to_ESR;

		X3 := S3;
		cnt := cnt + 1;
		esr_flag := TRUE;
	END_IF;
	IF cnt < 4 AND s4 <> X4 AND ((s4 < BYTE#100) OR (S4 > BYTE#99 AND S4 < BYTE#200 AND mode >= BYTE#2) OR (S4 > BYTE#199 AND mode = BYTE#3)) THEN

		status_to_ESR.status := s4;
		status_to_ESR.adress := a4;
		status_to_ESR.DT_in  := DT_in;
		status_to_ESR.TS     := tx;
		status_to_ESR();
		esr_out[cnt] := status_to_ESR.status_to_ESR;

		X4 := S4;
		cnt := cnt + 1;
		esr_flag := TRUE;
	END_IF;
	IF cnt < 4 AND s5 <> X5 AND ((s5 < BYTE#100) OR (S5 > BYTE#99 AND S5 < BYTE#200 AND mode >= BYTE#2) OR (S5 > BYTE#199 AND mode = BYTE#3)) THEN

		status_to_ESR.status := s5;
		status_to_ESR.adress := a5;
		status_to_ESR.DT_in  := DT_in;
		status_to_ESR.TS     := tx;
		status_to_ESR();
		esr_out[cnt] := status_to_ESR.status_to_ESR;

		X5 := S5;
		cnt := cnt + 1;
		esr_flag := TRUE;
	END_IF;
	IF cnt < 4 AND s6 <> X6 AND ((s6 < BYTE#100) OR (S6 > BYTE#99 AND S6 < BYTE#200 AND mode >= BYTE#2) OR (S6 > BYTE#199 AND mode = BYTE#3)) THEN

		status_to_ESR.status := s6;
		status_to_ESR.adress := a6;
		status_to_ESR.DT_in  := DT_in;
		status_to_ESR.TS     := tx;
		status_to_ESR();
		esr_out[cnt] := status_to_ESR.status_to_ESR;

		X6 := S6;
		cnt := cnt + 1;
		esr_flag := TRUE;
	END_IF;
	IF cnt < 4 AND s7 <> X7 AND ((s7 < BYTE#100) OR (S7 > BYTE#99 AND S7 < BYTE#200 AND mode >= BYTE#2) OR (S7 > BYTE#199 AND mode = BYTE#3)) THEN

		status_to_ESR.status := s7;
		status_to_ESR.adress := a7;
		status_to_ESR.DT_in  := DT_in;
		status_to_ESR.TS     := tx;
		status_to_ESR();
		esr_out[cnt] := status_to_ESR.status_to_ESR;

		X7 := S7;
		cnt := cnt + 1;
		esr_flag := TRUE;
	END_IF;

END_FUNCTION_BLOCK

PROGRAM program0

	VAR
	S0 :	BYTE;
	A0 :	STRING;
	S1 :	BYTE;
	A1 :	STRING;
	S2 :	BYTE;
	A2 :	STRING;
	S3 :	BYTE;
	A3 :	STRING;
	S4 :	BYTE;
	A4 :	STRING;
	S5 :	BYTE;
	A5 :	STRING;
	S6 :	BYTE;
	A6 :	STRING;
	S7 :	BYTE;
	A7 :	STRING;
	DT_IN :	UDINT;
	MODE :	BYTE;

	ESR_OUT :	oscat_ESR_3;

	ESR_FLAG :	BOOL;

		func_block : ESR_MON_X8;
  	END_VAR
	func_block.S0 := S0;
	func_block.A0 := A0;
	func_block.S1 := S1;
	func_block.A1 := A1;
	func_block.S2 := S2;
	func_block.A2 := A2;
	func_block.S3 := S3;
	func_block.A3 := A3;
	func_block.S4 := S4;
	func_block.A4 := A4;
	func_block.S5 := S5;
	func_block.A5 := A5;
	func_block.S6 := S6;
	func_block.A6 := A6;
	func_block.S7 := S7;
	func_block.A7 := A7;
	func_block.DT_IN := DT_IN;
	func_block.MODE := MODE;
	func_block.ESR_Out := ESR_Out;
	func_block();
	ESR_Out := func_block.ESR_Out;
	ESR_FLAG := func_block.ESR_FLAG;
END_PROGRAM

CONFIGURATION Config0

	VAR_GLOBAL
		PLC_TICKS_PER_SEC :	INT;
		PLC_SYS_TICK_CNT :	DINT;
	END_VAR

  	RESOURCE Res0 ON PLC
    	TASK task0(INTERVAL := T#20ms,PRIORITY := 0);
    	PROGRAM instance0 WITH task0 : program0;
  	END_RESOURCE

END_CONFIGURATION

(* ---- EVENTS.ST ---- *)
TYPE oscat_HOLIDAY_DATA :
  STRUCT
	NAME : STRING;
	DAY : SINT;
	MONTH : SINT;
	USE : SINT;
	PAD_BYTE : BYTE;
  END_STRUCT;
END_TYPE

TYPE
  oscat_HOLIDAY_DATA_0_29 	: ARRAY [0..29] OF oscat_HOLIDAY_DATA;
  oscat_HOLIDAY_DATA_0_49 	: ARRAY [0..49] OF oscat_HOLIDAY_DATA;
END_TYPE

FUNCTION DAY_OF_DATE:DINT
	VAR_INPUT
		IDATE :	UDINT;
	END_VAR

	day_of_date := UDINT_TO_DINT(idate / UDINT#86400);
END_FUNCTION

FUNCTION YEAR_OF_DATE:INT
	VAR_INPUT
		IDATE :	UDINT;
	END_VAR

	YEAR_OF_DATE := UDINT_TO_INT((idate+UDINT#43200) / UDINT#31557600 + UDINT#1970);
END_FUNCTION

FUNCTION _INT_TO_UDINT:UDINT
	VAR_INPUT
		IN :	INT;
	END_VAR

	_INT_TO_UDINT := DINT_TO_UDINT(INT_TO_DINT(IN));
END_FUNCTION

FUNCTION SET_DATE:UDINT

	VAR_INPUT
		YEAR :	INT;
		MONTH :	INT;
		DAY :	INT;
	END_VAR

	VAR
		count :	INT;
	END_VAR

	IF month > 2 THEN
		count := (month - 1) * 30;
		IF month > 7 THEN
			count := count + DWORD_TO_INT(SHR(DINT_TO_DWORD(INT_TO_DINT(month) - INT_TO_DINT(3)),1));
		ELSE
			count := count + DWORD_TO_INT(SHR(DINT_TO_DWORD(INT_TO_DINT(month) - INT_TO_DINT(4)),1));
		END_IF;
		IF SHL(INT_TO_WORD(year),14) = WORD#0 THEN
			count := count + 1;
		END_IF;
	ELSE
		count := (month - 1) * 31;
	END_IF;
	SET_DATE := (_INT_TO_UDINT(count + day - 1) + DWORD_TO_UDINT(SHR(UDINT_TO_DWORD(_INT_TO_UDINT(year) * UDINT#1461 - UDINT#2878169), 2))) * UDINT#86400;
END_FUNCTION

FUNCTION_BLOCK EVENTS
	VAR_INPUT
		DATE_IN :	UDINT;
		ENA :	BOOL;
	END_VAR

	VAR_OUTPUT
		Y :	BOOL;
		NAME :	STRING;
	END_VAR

	VAR_IN_OUT
		ELIST :	oscat_HOLIDAY_DATA_0_49;
	END_VAR

	VAR
		i :	INT;
		last_active :	UDINT;
		size :	INT := 49;
		day_in :	DINT;
		cyr :	INT;
		lday :	DINT;
		check :	oscat_HOLIDAY_DATA;
		y_int :	BOOL;
		name_int :	STRING;
	END_VAR

	IF last_active <> date_in THEN
		last_active := DATE_IN;
		Y_int := FALSE;
		name_int := '';
		day_in := DAY_OF_DATE(DATE_IN);
		cyr := YEAR_OF_DATE(DATE_IN);

		(* search list for events *)
		FOR i := 0 TO size DO
			check := elist[i];
			lday := DAY_OF_DATE(SET_DATE(cyr,SINT_TO_INT(check.month), SINT_TO_INT(check.day)));
			IF day_in >= lday AND day_in <= lday + SINT_TO_DINT(check.use) - DINT#1 THEN
				y_int := TRUE;
				name_int := check.name;
				EXIT;
			END_IF;
		END_FOR;
	END_IF;

	IF ENA THEN
		Y := y_int;
		NAME := name_int;
	ELSE
		Y := FALSE;
		NAME := '';
	END_IF;

END_FUNCTION_BLOCK

PROGRAM program0
	VAR
		DATE_IN :	UDINT;
		ENA :	BOOL;

		Y :	BOOL;
		NAME :	STRING;

		ELIST :	oscat_HOLIDAY_DATA_0_49;

		func_block : EVENTS;
	END_VAR
	func_block.DATE_IN := DATE_IN;
	func_block.ENA := ENA;
	func_block.ELIST := ELIST ;

	func_block();
	Y  := func_block.Y;
	NAME  := func_block.NAME;
	ELIST  := func_block.ELIST;
END_PROGRAM

CONFIGURATION Config0
	RESOURCE Res0 ON PLC
		TASK task0(INTERVAL := T#20ms,PRIORITY := 0);
		PROGRAM instance0 WITH task0 : program0;
	END_RESOURCE
END_CONFIGURATION

(* ---- F_LAMP.ST ---- *)
FUNCTION_BLOCK T_PLC_MS_block
	VAR_OUTPUT
		T_PLC_MS :	UDINT;
	END_VAR

	VAR_EXTERNAL
		PLC_TICKS_PER_SEC :	INT;
		PLC_SYS_TICK_CNT :	DINT;
	END_VAR

	VAR
		debug :	BOOL;(*Debug-Mode ON / OFF*)
		N :	INT;(*Debug-Faktor*)
		Offset :	UDINT;(*Debug-Offset*)
		temp :	DWORD := DWORD#1;(*Debug-Offset*)
		mode :	BOOL;(*modus*)
		faktor :	UDINT;(*Systemtakt-Faktor*)
		init :	BOOL;
		v_plc_ticks_per_sec :	UDINT;
		base :	UDINT := UDINT#1000;
	END_VAR

	IF init = FALSE THEN
		v_plc_ticks_per_sec := INT_TO_UDINT(PLC_TICKS_PER_SEC);
		IF v_plc_ticks_per_sec = UDINT#1024 THEN
			faktor := UDINT#1;
			mode := FALSE;
		ELSIF v_plc_ticks_per_sec > UDINT#0 THEN
			IF v_plc_ticks_per_sec <= base THEN
				faktor := base / v_plc_ticks_per_sec;
				mode := FALSE;
			ELSE
				faktor := v_plc_ticks_per_sec / base;
				mode := TRUE;
			END_IF;
		ELSE
			faktor := UDINT#1;
		END_IF;
		init := TRUE;
	END_IF;

	IF mode THEN
		T_PLC_MS := DINT_TO_UDINT(PLC_SYS_TICK_CNT) / faktor;
	ELSE
		T_PLC_MS := DINT_TO_UDINT(PLC_SYS_TICK_CNT) * faktor;
	END_IF;

	IF debug THEN
		T_PLC_MS := (DWORD_TO_UDINT(SHL(UDINT_TO_DWORD(T_PLC_MS),N) OR SHL(temp,N)) - UDINT#1) + Offset;
	END_IF;

END_FUNCTION_BLOCK

FUNCTION_BLOCK ONTIME_Block

	VAR_INPUT
		IN :	BOOL;
		RST :	BOOL;
	END_VAR

	VAR_IN_OUT
		SECONDS :	UDINT;
		CYCLES :	UDINT;
	END_VAR

	VAR
		tx :	UDINT;
		last :	UDINT;
		edge :	BOOL;
		init :	BOOL;
		ms :	UDINT;
		T_PLC_MS :	T_PLC_MS_Block;
	END_VAR

	T_PLC_MS();
	tx:= T_PLC_MS.T_PLC_MS;

	IF NOT init THEN
		init := TRUE;
		last := tx;
		ms := UDINT#0;
	END_IF;
	IF RST THEN
		SECONDS := UDINT#0;
		CYCLES := UDINT#0;
		last := tx;
		ms := UDINT#0;
	ELSIF IN THEN
		(* add the current milliseconds *)
		ms := (tx - last) + ms;
		IF ms >= UDINT#1000 THEN
			seconds := seconds + UDINT#1;
			ms := ms - UDINT#1000;
		END_IF;
		cycles := cycles + BOOL_TO_UDINT(NOT edge);
	END_IF;
	last := tx;
	edge := in;

END_FUNCTION_BLOCK

FUNCTION_BLOCK F_LAMP_Block

	VAR_INPUT
		SWITCH :	BOOL;
		DIMM :	BYTE := BYTE#255;
		RST :	BOOL;
		T_NO_DIMM :	UINT := UINT#100;
		T_MAINTENANCE :	UINT := UINT#15000;
	END_VAR

	VAR_OUTPUT
		LAMP :	BYTE;
		STATUS :	BYTE;
	END_VAR

	VAR_IN_OUT
		ONTIME :	UDINT;
		CYCLES :	UDINT;
	END_VAR

	VAR
		runtime :	ONTIME_Block;
	END_VAR

	runtime(in := switch, SECONDS := ONTIME , CYCLES := CYCLES);
	CYCLES := runtime.CYCLES;
	ONTIME := runtime.SECONDS;

	IF RST THEN
		ONTIME := UDINT#0;
		CYCLES := UDINT#0;
	END_IF;
	IF SWITCH THEN
		IF ontime < UINT_TO_UDINT(T_NO_DIMM) * UDINT#3600 THEN
			LAMP := BYTE#255;
			STATUS := BYTE#111;
		ELSE
			LAMP := DIMM;
			STATUS := BYTE#112;
		END_IF;
	ELSE
		LAMP := BYTE#0;
		STATUS := BYTE#110;
	END_IF;

	IF ontime >= UINT_TO_UDINT(T_maintenance) * UDINT#3600 AND T_Maintenance > UINT#0 THEN
		STATUS := BYTE#120;
	END_IF;

END_FUNCTION_BLOCK

PROGRAM program0
	VAR
	    SWITCH :	BOOL;
		DIMM :	BYTE := BYTE#255;
		RST :	BOOL;
		T_NO_DIMM :	UINT := UINT#100;
		T_MAINTENANCE :	UINT := UINT#15000;
		ONTIME :	UDINT;
		CYCLES :	UDINT;
		LAMP :	BYTE;
		STATUS :	BYTE;

		func_block : F_LAMP_Block;
  	END_VAR
	func_block.SWITCH := SWITCH;
	func_block.DIMM := DIMM;
	func_block.RST := RST;
	func_block.T_NO_DIMM := T_NO_DIMM;
	func_block.T_MAINTENANCE := T_MAINTENANCE;
	func_block.ONTIME := ONTIME;
	func_block.CYCLES := CYCLES;

	func_block();
	ONTIME := func_block.ONTIME;
	CYCLES := func_block.CYCLES;
	LAMP := func_block.LAMP;
	STATUS := func_block.STATUS;
END_PROGRAM

CONFIGURATION Config0
	VAR_GLOBAL
		PLC_TICKS_PER_SEC :	INT;
		PLC_SYS_TICK_CNT :	DINT;
	END_VAR
  	RESOURCE Res0 ON PLC
    	TASK task0(INTERVAL := T#20ms,PRIORITY := 0);
    	PROGRAM instance0 WITH task0 : program0;
  	END_RESOURCE
END_CONFIGURATION

(* ---- F_POLY.ST ---- *)
TYPE
  oscat_arr_0_7               : ARRAY [0..7]    OF REAL;
END_TYPE

FUNCTION_BLOCK F_POLY_Block
	VAR_INPUT
		X :	REAL;
		C :	oscat_arr_0_7;
	END_VAR

	VAR_OUTPUT
		F_POLY :	REAL;
	END_VAR

	F_POLY := ((((((( c[7] * x + c[6] ) * x + c[5] ) * x + c[4] ) * x + c[3] ) * x + c[2] ) * x + c[1] ) * x + c[0] ) ;

END_FUNCTION_BLOCK

PROGRAM program0
	VAR
		X :	REAL;
		C :	oscat_arr_0_7;

		F_POLY :	REAL;

		func_block : F_POLY_Block;
	END_VAR
	func_block.X := X;
	func_block.C := C;
	func_block();
	F_POLY  := func_block.F_POLY;
END_PROGRAM

CONFIGURATION Config0
	RESOURCE Res0 ON PLC
		TASK task0(INTERVAL := T#20ms,PRIORITY := 0);
		PROGRAM instance0 WITH task0 : program0;
	END_RESOURCE
END_CONFIGURATION

(* ---- FADE.ST ---- *)
FUNCTION_BLOCK T_PLC_MS_block
	VAR_OUTPUT
		T_PLC_MS :	UDINT;
	END_VAR

	VAR_EXTERNAL
		PLC_TICKS_PER_SEC :	INT;
		PLC_SYS_TICK_CNT :	DINT;
	END_VAR

	VAR
		debug :	BOOL;(*Debug-Mode ON / OFF*)
		N :	INT;(*Debug-Faktor*)
		Offset :	UDINT;(*Debug-Offset*)
		temp :	DWORD := DWORD#1;(*Debug-Offset*)
		mode :	BOOL;(*modus*)
		faktor :	UDINT;(*Systemtakt-Faktor*)
		init :	BOOL;
		v_plc_ticks_per_sec :	UDINT;
		base :	UDINT := UDINT#1000;
	END_VAR

	IF init = FALSE THEN
		v_plc_ticks_per_sec := INT_TO_UDINT(PLC_TICKS_PER_SEC);
		IF v_plc_ticks_per_sec = UDINT#1024 THEN
			faktor := UDINT#1;
			mode := FALSE;
		ELSIF v_plc_ticks_per_sec > UDINT#0 THEN
			IF v_plc_ticks_per_sec <= base THEN
				faktor := base / v_plc_ticks_per_sec;
				mode := FALSE;
			ELSE
				faktor := v_plc_ticks_per_sec / base;
				mode := TRUE;
			END_IF;
		ELSE
			faktor := UDINT#1;
		END_IF;
		init := TRUE;
	END_IF;

	IF mode THEN
		T_PLC_MS := DINT_TO_UDINT(PLC_SYS_TICK_CNT) / faktor;
	ELSE
		T_PLC_MS := DINT_TO_UDINT(PLC_SYS_TICK_CNT) * faktor;
	END_IF;

	IF debug THEN
		T_PLC_MS := (DWORD_TO_UDINT(SHL(UDINT_TO_DWORD(T_PLC_MS),N) OR SHL(temp,N)) - UDINT#1) + Offset;
	END_IF;
END_FUNCTION_BLOCK

FUNCTION _WORD_TO_DINT:DINT
	VAR_INPUT
		IN :	WORD;
	END_VAR
	_WORD_TO_DINT := UINT_TO_DINT(WORD_TO_UINT(IN));
END_FUNCTION

FUNCTION TIME_TO_UDINT2:UDINT
	VAR_INPUT
		X :	TIME;
	END_VAR

	TIME_TO_UDINT2 := DINT_TO_UDINT(TIME_TO_DINT(X));
END_FUNCTION

FUNCTION_BLOCK _RMP_W

	VAR_INPUT
		DIR :	BOOL;
		E :	BOOL := TRUE;
		TR :	TIME;
	END_VAR

	VAR_IN_OUT
		RMP :	WORD;
	END_VAR

	VAR
		T_PLC_MS :	T_PLC_MS_block;
		tx :	UDINT;
		tl :	UDINT;
		ptesss :	DINT;
		init :	BOOL;
		last_dir :	BOOL;
	END_VAR

	T_PLC_MS();
	tx := T_PLC_MS.T_PLC_MS;
	IF E AND init THEN
		(* we need to set tl = tx when direction changes *)
		IF dir XOR last_dir THEN
			tl := tx;
			last_dir := dir;
		END_IF;
		(* check_elapsed time and calculate only if necessary *)
		IF tr > t#0s THEN
			ptesss := DWORD_TO_DINT(UDINT_TO_DWORD(DWORD_TO_UDINT(SHL(UDINT_TO_DWORD(tx-tl), 16)) / TIME_TO_UDINT2(TR)));
		ELSE
			ptesss := DINT#65535;
		END_IF;
		IF ptesss > DINT#0 THEN
			(* perform the ptesss on the ramp *)
			tl := tx;
			(* calculate the ptesss response *)
			IF NOT dir THEN ptesss := - ptesss; END_IF;
			rmp := DINT_TO_WORD(LIMIT(DINT#0, _WORD_TO_DINT(rmp) + ptesss, DINT#65535));
		END_IF;
	ELSE
		tl := tx;
		init := TRUE;
	END_IF;
END_FUNCTION_BLOCK

FUNCTION_BLOCK RMP_W

	VAR_INPUT
		SET :	BOOL;
		PT :	TIME;
		E :	BOOL := TRUE;
		UP :	BOOL := TRUE;
		RST :	BOOL;
	END_VAR

	VAR_OUTPUT
		OUT :	WORD;
		BUSY :	BOOL;
		HIGH :	BOOL;
		LOW :	BOOL;
	END_VAR

	VAR
		rmp :	_RMP_W;
	END_VAR

	rmp(dir := UP, E := E, TR := PT, rmp := out);
	out := rmp.RMP;

	IF RST THEN
		out := WORD#0;
	ELSIF SET THEN
		out := WORD#65535;
	END_IF;

	low := out = WORD#0;
	high := out = WORD#65535;
	busy := NOT (low OR high) AND E;

END_FUNCTION_BLOCK

FUNCTION _WORD_TO_REAL:REAL
	VAR_INPUT
		IN :	WORD;
	END_VAR
	_WORD_TO_REAL := UINT_TO_REAL(WORD_TO_UINT(IN));
END_FUNCTION

FUNCTION_BLOCK FADE
	VAR_INPUT
		IN1 :	REAL;
		IN2 :	REAL;
		F :	BOOL;
		TF :	TIME;
		RST :	BOOL;
	END_VAR

	VAR_OUTPUT
		Y :	REAL;
	END_VAR

	VAR
		rmx :	RMP_W;
	END_VAR
	rmx(rst := rst AND NOT F, set := rst AND F, pt := TF, up := F);
	Y := (in2 - In1) / 65535.0 * _WORD_TO_REAL(rmx.out) + in1;

END_FUNCTION_BLOCK

PROGRAM program0
  VAR

	IN1 :	REAL;
	IN2 :	REAL;
	F   :	BOOL;
	TF  :	TIME;
	RST :	BOOL;

	Y :	REAL;

	func_block : FADE;
  END_VAR
	func_block.IN1 :=IN1;
	func_block.IN2 :=IN2;
	func_block.F   :=F  ;
	func_block.TF  :=TF ;
	func_block.RST :=RST;
	func_block();
	Y := func_block.Y;

END_PROGRAM

CONFIGURATION Config0
	VAR_GLOBAL
		PLC_TICKS_PER_SEC :	INT;
		PLC_SYS_TICK_CNT :	DINT;
	END_VAR
  	RESOURCE Res0 ON PLC
    	TASK task0(INTERVAL := T#20ms,PRIORITY := 0);
    	PROGRAM instance0 WITH task0 : program0;
  	END_RESOURCE
END_CONFIGURATION

(* ---- FF_D2E.ST ---- *)
FUNCTION_BLOCK FF_D2E
	VAR_INPUT
		D0 :	BOOL;
		D1 :	BOOL;
		CLK :	BOOL;
		RST :	BOOL;
	END_VAR

	VAR_OUTPUT
		Q0 :	BOOL;
		Q1 :	BOOL;
	END_VAR

	VAR
		edge :	BOOL;
	END_VAR

	IF rst THEN
		Q0 := FALSE;
		Q1 := FALSE;
	ELSIF clk AND NOT edge THEN
		Q0 := D0;
		Q1 := D1;
	END_IF;
	edge := CLK;

END_FUNCTION_BLOCK

PROGRAM program0
  VAR
	D0  :	BOOL;
	D1  :	BOOL;
	CLK :	BOOL;
	RST :	BOOL;

	Q0 :	BOOL;
	Q1 :	BOOL;

	func_block : FF_D2E;
  END_VAR
	func_block.D0  :=D0 ;
	func_block.D1  :=D1 ;
	func_block.CLK :=CLK;
	func_block.RST :=RST;
	func_block();
	Q0 := func_block.Q0;
	Q1 := func_block.Q1;
END_PROGRAM

CONFIGURATION Config0
  RESOURCE Res0 ON PLC
    TASK task0(INTERVAL := T#20ms,PRIORITY := 0);
    PROGRAM instance0 WITH task0 : program0;
  END_RESOURCE
END_CONFIGURATION

(* ---- FF_D4E.ST ---- *)
FUNCTION_BLOCK FF_D4E
	VAR_INPUT
		D0 :	BOOL;
		D1 :	BOOL;
		D2 :	BOOL;
		D3 :	BOOL;
		CLK :	BOOL;
		RST :	BOOL;
	END_VAR

	VAR_OUTPUT
		Q0 :	BOOL;
		Q1 :	BOOL;
		Q2 :	BOOL;
		Q3 :	BOOL;
	END_VAR

	VAR
		edge :	BOOL;
	END_VAR

	IF rst THEN
		Q0 := FALSE;
		Q1 := FALSE;
		Q2 := FALSE;
		Q3 := FALSE;
	ELSIF clk AND NOT edge THEN
		Q0 := D0;
		Q1 := D1;
		Q2 := D2;
		Q3 := D3;
	END_IF;
	edge := CLK;
END_FUNCTION_BLOCK

PROGRAM program0
  VAR
		D0  :	BOOL;
		D1  :	BOOL;
		D2  :	BOOL;
		D3  :	BOOL;
		CLK :	BOOL;
		RST :	BOOL;

		Q0 :	BOOL;
		Q1 :	BOOL;
		Q2 :	BOOL;
		Q3 :	BOOL;

	func_block : FF_D4E;
  END_VAR
	func_block.D0 :=D0 ;
	func_block.D1 :=D1 ;
	func_block.D2 :=D2 ;
	func_block.D3 :=D3 ;
	func_block.CLK:=CLK;
	func_block.RST:=RST;
	func_block();
	Q0 := func_block.Q0;
	Q1 := func_block.Q1;
	Q2 := func_block.Q2;
	Q3 := func_block.Q3;
END_PROGRAM

CONFIGURATION Config0
  RESOURCE Res0 ON PLC
    TASK task0(INTERVAL := T#20ms,PRIORITY := 0);
    PROGRAM instance0 WITH task0 : program0;
  END_RESOURCE
END_CONFIGURATION

(* ---- FF_DRE.ST ---- *)
FUNCTION_BLOCK FF_DRE
	VAR_INPUT
		SET :	BOOL;
		D :	BOOL;
		CLK :	BOOL;
		RST :	BOOL;
	END_VAR

	VAR_OUTPUT
		Q :	BOOL;
	END_VAR

	VAR
		edge :	BOOL;
	END_VAR

	IF rst OR set THEN
		Q := NOT rst;
	ELSIF clk AND NOT edge THEN
		Q := D;
	END_IF;
	edge := CLK;

END_FUNCTION_BLOCK

PROGRAM program0
  VAR
	SET :	BOOL;
	D   :	BOOL;
	CLK :	BOOL;
	RST :	BOOL;

	Q :	BOOL;

	func_block : FF_DRE;
  END_VAR
	func_block.SET:=SET;
	func_block.D  :=D  ;
	func_block.CLK:=CLK;
	func_block.RST:=RST;
	func_block();
	Q:= func_block.Q;
END_PROGRAM

CONFIGURATION Config0
  RESOURCE Res0 ON PLC
    TASK task0(INTERVAL := T#20ms,PRIORITY := 0);
    PROGRAM instance0 WITH task0 : program0;
  END_RESOURCE
END_CONFIGURATION

(* ---- FF_JKE.ST ---- *)
FUNCTION_BLOCK FF_JKE
	VAR_INPUT
		SET :	BOOL;
		J :	BOOL;
		CLK :	BOOL;
		K :	BOOL;
		RST :	BOOL;
	END_VAR

	VAR_OUTPUT
		Q :	BOOL;
	END_VAR

	VAR
		edge :	BOOL;
	END_VAR

	IF rst OR set THEN
		Q := NOT rst;
	ELSIF clk AND NOT edge THEN
		IF J XOR K THEN Q := J;
		ELSE Q := K XOR Q;
		END_IF;
	END_IF;
	edge := CLK;

END_FUNCTION_BLOCK

PROGRAM program0
  VAR
		SET :	BOOL;
		J   :	BOOL;
		CLK :	BOOL;
		K   :	BOOL;
		RST :	BOOL;

		Q :	BOOL;

	func_block : FF_JKE;
  END_VAR
	func_block.SET :=SET;
	func_block.J   :=J  ;
	func_block.CLK :=CLK;
	func_block.K   :=K  ;
	func_block.RST :=RST;
	func_block();
	Q := func_block.Q;
END_PROGRAM

CONFIGURATION Config0
  RESOURCE Res0 ON PLC
    TASK task0(INTERVAL := T#20ms,PRIORITY := 0);
    PROGRAM instance0 WITH task0 : program0;
  END_RESOURCE
END_CONFIGURATION

(* ---- FF_RSE.ST ---- *)
FUNCTION_BLOCK FF_RSE
	VAR_INPUT
		CS :	BOOL;
		CR :	BOOL;
		RST :	BOOL;
	END_VAR

	VAR_OUTPUT
		Q :	BOOL;
	END_VAR

	VAR
		es :	BOOL;
		er :	BOOL;
	END_VAR

	IF rst THEN
		(* asynchronous reset *)
		Q := FALSE;
	ELSIF CR AND NOT er THEN
		(* rising edge on CR *)
		Q := FALSE;
	ELSIF CS AND NOT es THEN
		(* rising edge on CS *)
		Q := TRUE;
	END_IF;

	es := CS;
	er := CR;
END_FUNCTION_BLOCK

PROGRAM program0
  VAR
	CS  :	BOOL;
	CR  :	BOOL;
	RST :	BOOL;

	Q :	BOOL;

	func_block : FF_RSE;
  END_VAR
	func_block.CS  :=CS ;
	func_block.CR  :=CR ;
	func_block.RST :=RST;
	func_block();
	Q := func_block.Q;
END_PROGRAM

CONFIGURATION Config0
  RESOURCE Res0 ON PLC
    TASK task0(INTERVAL := T#20ms,PRIORITY := 0);
    PROGRAM instance0 WITH task0 : program0;
  END_RESOURCE
END_CONFIGURATION

(* ---- FIFO_16.ST ---- *)
TYPE
	oscat_ardw_0_15             : ARRAY [0..15]   OF DWORD;
END_TYPE

FUNCTION INC1:INT

	VAR_INPUT
		X :	INT;
		N :	INT;
	END_VAR

	IF X >= N - 1 THEN
		INC1 := 0;
	ELSE
		INC1 := X + 1;
	END_IF;
END_FUNCTION

FUNCTION_BLOCK FIFO_16
	VAR_INPUT
		DIN :	DWORD;
		E :	BOOL := TRUE;
		RD :	BOOL;
		WD :	BOOL;
		RST :	BOOL;
	END_VAR

	VAR_OUTPUT
		DOUT :	DWORD;
		EMPTY :	BOOL := TRUE;
		FULL :	BOOL;
	END_VAR

	VAR
		fifo :	oscat_ardw_0_15;
		pr :	INT;
		pw :	INT;
	END_VAR

	IF RST THEN
		pw := pr;
		FULL := FALSE;
		EMPTY := TRUE;
		Dout := DWORD#0;
	ELSIF E THEN
		IF NOT EMPTY AND RD THEN
			Dout := fifo[pr];
			pr := INC1(pr,16);
			EMPTY := pr = pw;
			FULL := FALSE;
		END_IF;
		IF NOT FULL AND WD THEN
			fifo[pw] := Din;
			pw := INC1(pw,16);
			FULL := pw = pr;
			EMPTY := FALSE;
		END_IF;
	END_IF;
END_FUNCTION_BLOCK

PROGRAM program0
  VAR
	DIN :	DWORD;
	E   :	BOOL;
	RD  :	BOOL;
	WD  :	BOOL;
	RST :	BOOL;

	DOUT  :	DWORD;
	EMPTY :	BOOL;
	FULL  :	BOOL;

	func_block : FIFO_16;
  END_VAR
	func_block.DIN :=DIN;
	func_block.E   :=E  ;
	func_block.RD  :=RD ;
	func_block.WD  :=WD ;
	func_block.RST :=RST;
	func_block();
	DOUT := func_block.DOUT ;
	EMPTY:= func_block.EMPTY;
	FULL := func_block.FULL ;
END_PROGRAM

CONFIGURATION Config0
  RESOURCE Res0 ON PLC
    TASK task0(INTERVAL := T#20ms,PRIORITY := 0);
    PROGRAM instance0 WITH task0 : program0;
  END_RESOURCE
END_CONFIGURATION

(* ---- FIFO_32.ST ---- *)
TYPE
	oscat_ardw_0_31             : ARRAY [0..31]   OF DWORD;
END_TYPE

FUNCTION INC1:INT

	VAR_INPUT
		X :	INT;
		N :	INT;
	END_VAR

	IF X >= N - 1 THEN
		INC1 := 0;
	ELSE
		INC1 := X + 1;
	END_IF;
END_FUNCTION

FUNCTION_BLOCK FIFO_32

	VAR_INPUT
		DIN :	DWORD;
		E :	BOOL := TRUE;
		RD :	BOOL;
		WD :	BOOL;
		RST :	BOOL;
	END_VAR

	VAR_OUTPUT
		DOUT :	DWORD;
		EMPTY :	BOOL := TRUE;
		FULL :	BOOL;
	END_VAR

	VAR
		fifo :	oscat_ardw_0_31;
		pr :	INT;
		pw :	INT;
	END_VAR

	IF RST THEN
		pw := pr;
		FULL := FALSE;
		EMPTY := TRUE;
		Dout := DWORD#0;
	ELSIF E THEN
		IF NOT EMPTY AND RD THEN
			Dout := fifo[pr];
			pr := INC1(pr,32);
			EMPTY := pr = pw;
			FULL := FALSE;
		END_IF;
		IF NOT FULL AND WD THEN
			fifo[pw] := Din;
			pw := INC1(pw,32);
			FULL := pw = pr;
			EMPTY := FALSE;
		END_IF;
	END_IF;

END_FUNCTION_BLOCK

PROGRAM program0
  VAR
	DIN :	DWORD;
	E   :	BOOL;
	RD  :	BOOL;
	WD  :	BOOL;
	RST :	BOOL;

	DOUT  :	DWORD;
	EMPTY :	BOOL;
	FULL  :	BOOL;

	func_block : FIFO_32;
  END_VAR
	func_block.DIN :=DIN;
	func_block.E   :=E  ;
	func_block.RD  :=RD ;
	func_block.WD  :=WD ;
	func_block.RST :=RST;
	func_block();
	DOUT := func_block.DOUT ;
	EMPTY:= func_block.EMPTY;
	FULL := func_block.FULL ;
END_PROGRAM

CONFIGURATION Config0
  RESOURCE Res0 ON PLC
    TASK task0(INTERVAL := T#20ms,PRIORITY := 0);
    PROGRAM instance0 WITH task0 : program0;
  END_RESOURCE
END_CONFIGURATION

(* ---- FILE_BLOCK.ST ---- *)
TYPE
  oscat_FILE_SERVER_DATA : STRUCT
	FILE_OPEN	: BOOL;
    FILENAME 	: STRING;
    MODE	 	: BYTE;
    OFFSET   	: UDINT;
    FILE_SIZE   : UDINT;
    AUTO_CLOSE	: TIME;
    ERROR	 	: BYTE;
  END_STRUCT;

  oscat_NW_BUF_LONG  : ARRAY [0..4095] OF BYTE;
  oscat_NETWORK_BUFFER :
  STRUCT
    SIZE   : UINT;
    BUFFER : oscat_NW_BUF_LONG;
  END_STRUCT;
END_TYPE

FUNCTION_BLOCK FILE_BLOCK

	VAR_IN_OUT
		MODE :	BYTE;
		FILENAME :	STRING;
		FSD :	oscat_FILE_SERVER_DATA;
		PT :	oscat_NETWORK_BUFFER;
	END_VAR

	VAR_INPUT
		POS :	UDINT;
	END_VAR

	VAR_OUTPUT
		ERROR :	BYTE;
		DATA :	BYTE;
	END_VAR

	VAR
		stepp :	INT;
		i :	INT;
		data_start :	UDINT;
		data_stop :	UDINT;
	END_VAR

	CASE stepp OF
	0:	IF MODE > BYTE#0 THEN
			ERROR := BYTE#0;
			IF FSD.FILE_OPEN AND (FSD.FILE_SIZE = UDINT#0 OR POS >= FSD.FILE_SIZE) THEN
				ERROR := BYTE#255;
				MODE := BYTE#0;
			ELSIF POS < data_start OR POS > data_stop OR NOT FSD.FILE_OPEN THEN
				FSD.FILENAME := FILENAME;
				FSD.MODE := BYTE#1;
				FSD.OFFSET := POS;
				PT.SIZE := UINT#65535;
				data_start := UDINT#0;
				data_stop := UDINT#0;
				stepp := 10;
			ELSE
				i := UDINT_TO_INT(POS - data_start);
				DATA := PT.BUFFER[i];
				MODE := BYTE#0;
			END_IF;
		END_IF;

	10:	IF FSD.MODE = BYTE#0 THEN
			IF FSD.ERROR > BYTE#0 THEN
				ERROR := FSD.ERROR;
				MODE := BYTE#0;
			ELSE
				data_start := POS;
				data_stop := POS + UINT_TO_UDINT(PT.SIZE) - UDINT#1;
			END_IF;
			stepp := 0;
		END_IF;
	END_CASE;
END_FUNCTION_BLOCK

PROGRAM program0
	VAR
		MODE :	BYTE;
		FILENAME :	STRING;
		FSD :	oscat_FILE_SERVER_DATA;
		PT :	oscat_NETWORK_BUFFER;
		POS :	UDINT;
		ERROR :	BYTE;
		DATA :	BYTE;

		func_block : FILE_BLOCK;
	END_VAR
	func_block.MODE    :=MODE    ;
	func_block.FILENAME:=FILENAME;
	func_block.FSD     :=FSD     ;
	func_block.PT      :=PT      ;
	func_block.POS     :=POS     ;
	func_block();
	MODE    := func_block.MODE    ;
	FILENAME:= func_block.FILENAME;
	FSD     := func_block.FSD     ;
	PT      := func_block.PT      ;
	ERROR   := func_block.ERROR;
	DATA    := func_block.DATA;

END_PROGRAM

CONFIGURATION Config0
  RESOURCE Res0 ON PLC
    TASK task0(INTERVAL := T#20ms,PRIORITY := 0);
    PROGRAM instance0 WITH task0 : program0;
  END_RESOURCE
END_CONFIGURATION

(* ---- FILE_PATH_SPLIT.ST ---- *)
TYPE
  oscat_STRING250             : STRING;
  oscat_STRING1             : STRING;
  oscat_STRING80             : STRING;
  oscat_STRING3             : STRING;
  oscat_NW_BUF_LONG  : ARRAY [0..4095] OF BYTE;
  PRINTF_DATA_250  	:  ARRAY [1..11]  OF oscat_STRING250;
  PRINTF_DATA_80 	:  ARRAY [1..11]  OF oscat_STRING80;
  LOG_250       	:  ARRAY [0..400] OF oscat_STRING250;
  LOG_80    		:  ARRAY [0..400] OF oscat_STRING80;
  LOG_OPTION		:  ARRAY [0..400] OF DWORD;

  us_LOG_CONTROL :
  STRUCT
    NEW_MSG              : oscat_STRING250;    (*W neue Nachricht f�r den Datenbuffer   *)
	NEW_MSG_OPTION 		 : DWORD;
    LEVEL                : BYTE;
	SIZE                 : INT;                (*R Anzahl der Strings im LOG_DATA       *)
	RESET                : BOOL;               (*W Nachrichtenbuffer l�schen            *)
    PRINTF               : PRINTF_DATA_250;    (*W Array PRINTF Parameter               *)
    MSG                  : LOG_250;            (*I Array Message                        *)
    MSG_OPTION           : LOG_OPTION;     	   (*I Array Message Option                 *)
	UPDATE_COUNT         : UINT;               (*R Updatez�hler                         *)
    IDX                  : INT;                (*R aktueller Nachrichten-Index          *)
	RING_MODE            : BOOL;               (*I Buffer�berlauf erkannt               *)
  END_STRUCT;

  us_LOG_CONTROL_80 :
  STRUCT
    NEW_MSG              : oscat_STRING80;     (*W neue Nachricht f�r den Datenbuffer   *)
	NEW_MSG_OPTION 		 : DWORD;
    LEVEL                : BYTE;
	SIZE                 : INT;                (*R Anzahl der Strings im LOG_DATA       *)
	RESET                : BOOL;               (*W Nachrichtenbuffer l�schen            *)
    PRINTF               : PRINTF_DATA_80;     (*W Array PRINTF Parameter               *)
    MSG                  : LOG_80;             (*I Array Message                        *)
    MSG_OPTION           : LOG_OPTION;     	   (*I Array Message Option                 *)
	UPDATE_COUNT         : UINT;               (*R Updatez�hler                         *)
    IDX                  : INT;                (*R aktueller Nachrichten-Index          *)
	RING_MODE            : BOOL;               (*I Buffer�berlauf erkannt               *)
  END_STRUCT;

  LINE_ARRAY 			: ARRAY [1..40] OF INT;

  us_LOG_VIEWPORT :
    STRUCT
     LINE_ARRAY          : LINE_ARRAY;
     COUNT               : INT;                (* Anzahl der sichtbaren Nachtrichten   *)
	 UPDATE_COUNT        : UINT;               (* Updatez�hler                         *)
     MOVE_TO_X           : INT;                (* Steuerung der Nachrichtenanzeige     *)
     UPDATE              : BOOL;               (* Daten wurden ge�ndert -> neuzeichnen *)
  END_STRUCT;

  oscat_FILE_SERVER_DATA : STRUCT
	FILE_OPEN	: BOOL;
    FILENAME 	: STRING;
    MODE	 	: BYTE;
    OFFSET   	: UDINT;
    FILE_SIZE   : UDINT;
    AUTO_CLOSE	: TIME;
    ERROR	 	: BYTE;
  END_STRUCT;

  oscat_FILE_PATH_DATA : STRUCT
	DRIVE : oscat_string3;
	DIRECTORY : oscat_string250;
	FILENAME : STRING;
  END_STRUCT;

  oscat_UNI_CIRCULAR_BUFFER_DATA : STRUCT
	D_MODE : INT;
	D_HEAD : WORD;
	D_STRING : oscat_string250;
	D_REAL : REAL;
	D_DWORD : DWORD;
	BUF_SIZE : INT;
	BUF_COUNT : INT;
	BUF_USED : USINT;
	BUF : oscat_NW_BUF_LONG;
	_GetStart : INT;
	_GetEnd : INT;
	_Last : INT;
	_First : INT;
  END_STRUCT;

  oscat_DLOG_DATA : STRUCT
	STORE_TYPE : BYTE;
	ADD_HEADER : BOOL;
	ADD_DATA : BOOL;
	ADD_DATA_REQ : BOOL;
	CLOCK_TRIG : BOOL;
	ID_MAX : USINT;
	DTI : UDINT;
	UCB : oscat_UNI_CIRCULAR_BUFFER_DATA;
	NEW_FILE : STRING;
	NEW_FILE_RTRIG : BOOL;
  END_STRUCT;

END_TYPE

FUNCTION_BLOCK FILE_PATH_SPLIT_Block

	VAR_INPUT
		FILENAME :	oscat_STRING250;
	END_VAR

	VAR_OUTPUT
		FILE_PATH_SPLIT :	BOOL;
	END_VAR

	VAR_IN_OUT
		X :	oscat_FILE_PATH_DATA;
	END_VAR

	VAR
		b :	INT;
		c :	INT;
		d :	oscat_STRING1;
		p1 :	INT;
		p2 :	INT;
	END_VAR

	X.DRIVE := '';
	X.DIRECTORY := '';
	X.FILENAME := '';
	p1 := 0;
	p2 := 0;
	c := LEN(FILENAME);
	IF c = 0 THEN
		FILE_PATH_SPLIT := FALSE;
		RETURN;
	END_IF;

	FOR b := 1 TO c DO
		d := MID(FILENAME, 1, b);
		IF EQ_STRING(d,':') THEN
			p1 := b;
		ELSIF EQ_STRING(d,'/') OR EQ_STRING(d,'\') THEN
			p2 := b;
		END_IF;
	END_FOR;

	IF p1 = 2 THEN
		X.DRIVE := LEFT(FILENAME,p1);
	END_IF;

	IF p2 > 0 AND p2 > p1 THEN
		X.DIRECTORY := MID(FILENAME,p2-p1,p1+1);
	END_IF;

	X.FILENAME := RIGHT(FILENAME,c - MAX (p1,p2));
	FILE_PATH_SPLIT := TRUE;

END_FUNCTION_BLOCK

PROGRAM program0
	VAR
		FILENAME :	oscat_STRING250;
		FILE_PATH_SPLIT :	BOOL;
		X :	oscat_FILE_PATH_DATA;

		func_block : FILE_PATH_SPLIT_Block;
	END_VAR
	func_block.FILENAME := FILENAME;
	func_block.X := X;

	func_block();
	FILE_PATH_SPLIT  := func_block.FILE_PATH_SPLIT;
	X  := func_block.X;
END_PROGRAM

CONFIGURATION Config0
	RESOURCE Res0 ON PLC
		TASK task0(INTERVAL := T#20ms,PRIORITY := 0);
		PROGRAM instance0 WITH task0 : program0;
	END_RESOURCE
END_CONFIGURATION

(* ---- FILL.ST ---- *)
FUNCTION_BLOCK CHR_TO_STRING_Block
	VAR_INPUT
		C :	BYTE;
	END_VAR

	VAR_OUTPUT
		CHR_TO_STRING :	STRING;
	END_VAR

	CHR_TO_STRING := BYTE_TO_STRING(C);

END_FUNCTION_BLOCK

FUNCTION BIT_OF_DWORD : BOOL
  VAR_INPUT
    IN : DWORD;
    N : INT;
  END_VAR

  BIT_OF_DWORD := (SHR(in,N) AND 16#00000001) > 0;
  (* from OSCAT library; www.oscat.de  *)
END_FUNCTION

FUNCTION_BLOCK FILL_Block
	VAR_INPUT
		C :	BYTE;
		L :	INT;
	END_VAR

	VAR_OUTPUT
		FILL :	STRING;
	END_VAR

	VAR
		N :	BYTE;
		I :	INT;
		sx :	STRING;
		CHR_TO_STRING :	CHR_TO_STRING_Block;
		FILL_tmp :	STRING;
	END_VAR

	CHR_TO_STRING(C:=c);
	Sx:=CHR_TO_STRING.CHR_TO_STRING;
	(* create string *)
	N := INT_TO_BYTE(LIMIT(0,L,80));
	(* create a string of characters to be connected to str *)
	FILL := '';
	FOR i := 1 TO 8 DO
		FILL_tmp := FILL;
		FILL := CONCAT(FILL_tmp,FILL);
		IF BIT_OF_DWORD(BYTE_TO_DWORD(N),7) THEN FILL := CONCAT(FILL,Sx); END_IF;
		N := SHL(N,1);
	END_FOR;
END_FUNCTION_BLOCK

PROGRAM program0
  VAR
	C :	BYTE;
	L :	INT;

	FILL :	STRING;

	func_block : FILL_Block;
  END_VAR
	func_block.C  :=C ;
	func_block.L  :=L ;
	func_block();
	FILL := func_block.FILL;
END_PROGRAM

CONFIGURATION Config0
  RESOURCE Res0 ON PLC
    TASK task0(INTERVAL := T#20ms,PRIORITY := 0);
    PROGRAM instance0 WITH task0 : program0;
  END_RESOURCE
END_CONFIGURATION

(* ---- FILTER_DW.ST ---- *)
FUNCTION_BLOCK T_PLC_MS_block
	VAR_OUTPUT
		T_PLC_MS :	UDINT;
	END_VAR

	VAR_EXTERNAL
		PLC_TICKS_PER_SEC :	INT;
		PLC_SYS_TICK_CNT :	DINT;
	END_VAR

	VAR
		debug :	BOOL;(*Debug-Mode ON / OFF*)
		N :	INT;(*Debug-Faktor*)
		Offset :	UDINT;(*Debug-Offset*)
		temp :	DWORD := DWORD#1;(*Debug-Offset*)
		mode :	BOOL;(*modus*)
		faktor :	UDINT;(*Systemtakt-Faktor*)
		init :	BOOL;
		v_plc_ticks_per_sec :	UDINT;
		base :	UDINT := UDINT#1000;
	END_VAR

	IF init = FALSE THEN
		v_plc_ticks_per_sec := INT_TO_UDINT(PLC_TICKS_PER_SEC);
		IF v_plc_ticks_per_sec = UDINT#1024 THEN
			faktor := UDINT#1;
			mode := FALSE;
		ELSIF v_plc_ticks_per_sec > UDINT#0 THEN
			IF v_plc_ticks_per_sec <= base THEN
				faktor := base / v_plc_ticks_per_sec;
				mode := FALSE;
			ELSE
				faktor := v_plc_ticks_per_sec / base;
				mode := TRUE;
			END_IF;
		ELSE
			faktor := UDINT#1;
		END_IF;
		init := TRUE;
	END_IF;

	IF mode THEN
		T_PLC_MS := DINT_TO_UDINT(PLC_SYS_TICK_CNT) / faktor;
	ELSE
		T_PLC_MS := DINT_TO_UDINT(PLC_SYS_TICK_CNT) * faktor;
	END_IF;

	IF debug THEN
		T_PLC_MS := (DWORD_TO_UDINT(SHL(UDINT_TO_DWORD(T_PLC_MS),N) OR SHL(temp,N)) - UDINT#1) + Offset;
	END_IF;

END_FUNCTION_BLOCK

FUNCTION _DWORD_TO_REAL:REAL
	VAR_INPUT
		IN :	DWORD;
	END_VAR

	_DWORD_TO_REAL := UDINT_TO_REAL(DWORD_TO_UDINT(IN));
END_FUNCTION

FUNCTION _REAL_TO_DWORD: DWORD

  VAR_INPUT
    X :	REAL;
  END_VAR

  IF REAL_TO_DWORD(0.5) = DWORD#1 THEN
    _REAL_TO_DWORD := REAL_TO_DWORD(x);
  ELSIF X > 0.0 THEN
    _REAL_TO_DWORD := REAL_TO_DWORD(x+0.5);
  ELSIF X < 0.0 THEN
    _REAL_TO_DWORD := REAL_TO_DWORD(x-0.5);
  ELSE
    _REAL_TO_DWORD := DWORD#0;
  END_IF;
END_FUNCTION

FUNCTION_BLOCK FILTER_DW

	VAR_INPUT
		X :	DWORD;
		T :	TIME;
	END_VAR

	VAR_OUTPUT
		Y :	DWORD;
	END_VAR

	VAR
		last :	UDINT;
		tx :	UDINT;
		init :	BOOL;
		Yi :	REAL;
		T_PLC_MS :	T_PLC_MS_block;
	END_VAR

	T_PLC_MS();
	tx:= T_PLC_MS.T_PLC_MS;

	IF NOT init OR T = t#0s THEN
		init := TRUE;
		Yi := _DWORD_TO_REAL(X);
	ELSE
		Yi := Yi + (_DWORD_TO_REAL(X) - _DWORD_TO_REAL(Y)) * UDINT_TO_REAL(tx - last) / TIME_TO_REAL(T);
	END_IF;
	last := tx;

	Y := _REAL_TO_DWORD(Yi);

END_FUNCTION_BLOCK

PROGRAM program0
  VAR
	X :	DWORD;
	T :	TIME;

	Y :	DWORD;

	func_block : FILTER_DW;
  END_VAR
	func_block.X  := X;
	func_block.T  := T;
	func_block();
	Y := func_block.Y;
END_PROGRAM

CONFIGURATION Config0
	VAR_GLOBAL
		PLC_TICKS_PER_SEC :	INT;
		PLC_SYS_TICK_CNT :	DINT;
	END_VAR
	RESOURCE Res0 ON PLC
		TASK task0(INTERVAL := T#20ms,PRIORITY := 0);
		PROGRAM instance0 WITH task0 : program0;
	END_RESOURCE
END_CONFIGURATION

(* ---- FILTER_I.ST ---- *)
FUNCTION_BLOCK T_PLC_MS_block
	VAR_OUTPUT
		T_PLC_MS :	UDINT;
	END_VAR

	VAR_EXTERNAL
		PLC_TICKS_PER_SEC :	INT;
		PLC_SYS_TICK_CNT :	DINT;
	END_VAR

	VAR
		debug :	BOOL;(*Debug-Mode ON / OFF*)
		N :	INT;(*Debug-Faktor*)
		Offset :	UDINT;(*Debug-Offset*)
		temp :	DWORD := DWORD#1;(*Debug-Offset*)
		mode :	BOOL;(*modus*)
		faktor :	UDINT;(*Systemtakt-Faktor*)
		init :	BOOL;
		v_plc_ticks_per_sec :	UDINT;
		base :	UDINT := UDINT#1000;
	END_VAR

	IF init = FALSE THEN
		v_plc_ticks_per_sec := INT_TO_UDINT(PLC_TICKS_PER_SEC);
		IF v_plc_ticks_per_sec = UDINT#1024 THEN
			faktor := UDINT#1;
			mode := FALSE;
		ELSIF v_plc_ticks_per_sec > UDINT#0 THEN
			IF v_plc_ticks_per_sec <= base THEN
				faktor := base / v_plc_ticks_per_sec;
				mode := FALSE;
			ELSE
				faktor := v_plc_ticks_per_sec / base;
				mode := TRUE;
			END_IF;
		ELSE
			faktor := UDINT#1;
		END_IF;
		init := TRUE;
	END_IF;

	IF mode THEN
		T_PLC_MS := DINT_TO_UDINT(PLC_SYS_TICK_CNT) / faktor;
	ELSE
		T_PLC_MS := DINT_TO_UDINT(PLC_SYS_TICK_CNT) * faktor;
	END_IF;

	IF debug THEN
		T_PLC_MS := (DWORD_TO_UDINT(SHL(UDINT_TO_DWORD(T_PLC_MS),N) OR SHL(temp,N)) - UDINT#1) + Offset;
	END_IF;

END_FUNCTION_BLOCK

FUNCTION_BLOCK FILTER_I
	VAR_INPUT
		X :	INT;
		T :	TIME;
	END_VAR

	VAR_OUTPUT
		Y :	INT;
	END_VAR

	VAR
		Yi :	DINT;
		last :	UDINT;
		tx :	UDINT;
		init :	BOOL;
		T_PLC_MS :	T_PLC_MS_block;
	END_VAR

	T_PLC_MS();
	tx:= T_PLC_MS.T_PLC_MS;

	IF NOT init OR T = t#0s THEN
		init := TRUE;
		Yi := INT_TO_DINT(X) * DINT#1000;
	ELSE
		Yi := Yi + INT_TO_DINT(X - Y) * UDINT_TO_DINT(tx - last) * DINT#1000 / TIME_TO_DINT(T);
	END_IF;
	last := tx;
	Y := DINT_TO_INT(yi / DINT#1000);

END_FUNCTION_BLOCK

PROGRAM program0
  VAR
	X :	INT;
	T :	TIME;

	Y :	INT;

	func_block : FILTER_I;
  END_VAR
	func_block.X  := X;
	func_block.T  := T;
	func_block();
	Y := func_block.Y;
END_PROGRAM

CONFIGURATION Config0
	VAR_GLOBAL
		PLC_TICKS_PER_SEC :	INT;
		PLC_SYS_TICK_CNT :	DINT;
	END_VAR
	RESOURCE Res0 ON PLC
		TASK task0(INTERVAL := T#20ms,PRIORITY := 0);
		PROGRAM instance0 WITH task0 : program0;
	END_RESOURCE
END_CONFIGURATION

(* ---- FILTER_MAV_DW.ST ---- *)
TYPE
  oscat_ardw_0_31             : ARRAY [0..31]   OF DWORD;
END_TYPE

FUNCTION INC1:INT

	VAR_INPUT
		X :	INT;
		N :	INT;
	END_VAR

	IF X >= N - 1 THEN
		INC1 := 0;
	ELSE
		INC1 := X + 1;
	END_IF;
END_FUNCTION

FUNCTION_BLOCK FILTER_MAV_DW

	VAR_INPUT
		X :	DWORD;
		N :	UINT;
		RST :	BOOL;
	END_VAR

	VAR_OUTPUT
		Y :	DWORD;
	END_VAR

	VAR
		init :	BOOL;
		buffer :	oscat_ardw_0_31;
		i :	INT;
		tmp :	INT;
	END_VAR

	N := MIN(N, UINT#32);

	(* startup initialisation *)
	IF NOT init OR rst OR N = UINT#0 THEN
		init := TRUE;
		tmp := UINT_TO_INT(N)-1;
		FOR i := 0 TO tmp DO
			buffer[i] := X;
		END_FOR;
		Y := X;
	ELSE
		tmp := UINT_TO_INT(N);
		i := INC1(i, tmp);
		Y := UDINT_TO_DWORD(DWORD_TO_UDINT(Y) + (DWORD_TO_UDINT(X) - DWORD_TO_UDINT(buffer[i])) / UINT_TO_UDINT(N));
		buffer[i] := X;
	END_IF;

END_FUNCTION_BLOCK

PROGRAM program0
  VAR
	X :	DWORD;
	N :	UINT;
	RST :	BOOL;

	Y :	DWORD;

	func_block : FILTER_MAV_DW;
  END_VAR
	func_block.X  := X;
	func_block.N  := N;
	func_block.RST  := RST;
	func_block();
	Y := func_block.Y;
END_PROGRAM

CONFIGURATION Config0

	RESOURCE Res0 ON PLC
		TASK task0(INTERVAL := T#20ms,PRIORITY := 0);
		PROGRAM instance0 WITH task0 : program0;
	END_RESOURCE
END_CONFIGURATION

(* ---- FILTER_MAV_W.ST ---- *)
TYPE
  oscat_FILTER_MAV_W          : ARRAY [0..31]   OF WORD;
END_TYPE

FUNCTION INC1:INT

	VAR_INPUT
		X :	INT;
		N :	INT;
	END_VAR

	IF X >= N - 1 THEN
		INC1 := 0;
	ELSE
		INC1 := X + 1;
	END_IF;
END_FUNCTION

FUNCTION_BLOCK FILTER_MAV_W
	VAR_INPUT
		X :	WORD;
		N :	UINT;
		RST :	BOOL;
	END_VAR

	VAR_OUTPUT
		Y :	WORD;
	END_VAR

	VAR
		init :	BOOL;
		buffer :	oscat_FILTER_MAV_W;
		i :	INT;
		sum :	UDINT;
		tmp :	INT;
	END_VAR

	N := MIN(N, UINT#32);

	(* startup initialisation *)
	IF NOT init OR rst OR N = UINT#0 THEN
		init := TRUE;
		tmp := UINT_TO_INT(N) - 1;
		FOR i := 1 TO tmp DO
			buffer[i] := X;
		END_FOR;
		sum := UINT_TO_UDINT(WORD_TO_UINT(Y) * N);
		Y := X;
	ELSE
		tmp := UINT_TO_INT(N);
		i := INC1(i, tmp);
		sum := sum + WORD_TO_UDINT(X) - WORD_TO_UDINT(buffer[i]);
		Y := UDINT_TO_WORD(sum / UINT_TO_UDINT(N));
		buffer[i] := X;
	END_IF;

END_FUNCTION_BLOCK

PROGRAM program0
  VAR
	X :	WORD;
	N :	UINT;
	RST :	BOOL;

	Y :	WORD;

	func_block : FILTER_MAV_W;
  END_VAR
	func_block.X  := X;
	func_block.N  := N;
	func_block.RST  := RST;
	func_block();
	Y := func_block.Y;
END_PROGRAM

CONFIGURATION Config0

	RESOURCE Res0 ON PLC
		TASK task0(INTERVAL := T#20ms,PRIORITY := 0);
		PROGRAM instance0 WITH task0 : program0;
	END_RESOURCE
END_CONFIGURATION

(* ---- FILTER_W.ST ---- *)
FUNCTION_BLOCK T_PLC_MS_block
	VAR_OUTPUT
		T_PLC_MS :	UDINT;
	END_VAR

	VAR_EXTERNAL
		PLC_TICKS_PER_SEC :	INT;
		PLC_SYS_TICK_CNT :	DINT;
	END_VAR

	VAR
		debug :	BOOL;(*Debug-Mode ON / OFF*)
		N :	INT;(*Debug-Faktor*)
		Offset :	UDINT;(*Debug-Offset*)
		temp :	DWORD := DWORD#1;(*Debug-Offset*)
		mode :	BOOL;(*modus*)
		faktor :	UDINT;(*Systemtakt-Faktor*)
		init :	BOOL;
		v_plc_ticks_per_sec :	UDINT;
		base :	UDINT := UDINT#1000;
	END_VAR

	IF init = FALSE THEN
		v_plc_ticks_per_sec := INT_TO_UDINT(PLC_TICKS_PER_SEC);
		IF v_plc_ticks_per_sec = UDINT#1024 THEN
			faktor := UDINT#1;
			mode := FALSE;
		ELSIF v_plc_ticks_per_sec > UDINT#0 THEN
			IF v_plc_ticks_per_sec <= base THEN
				faktor := base / v_plc_ticks_per_sec;
				mode := FALSE;
			ELSE
				faktor := v_plc_ticks_per_sec / base;
				mode := TRUE;
			END_IF;
		ELSE
			faktor := UDINT#1;
		END_IF;
		init := TRUE;
	END_IF;

	IF mode THEN
		T_PLC_MS := DINT_TO_UDINT(PLC_SYS_TICK_CNT) / faktor;
	ELSE
		T_PLC_MS := DINT_TO_UDINT(PLC_SYS_TICK_CNT) * faktor;
	END_IF;

	IF debug THEN
		T_PLC_MS := (DWORD_TO_UDINT(SHL(UDINT_TO_DWORD(T_PLC_MS),N) OR SHL(temp,N)) - UDINT#1) + Offset;
	END_IF;

END_FUNCTION_BLOCK

FUNCTION_BLOCK FILTER_W
	VAR_INPUT
		X :	WORD;
		T :	TIME;
	END_VAR

	VAR_OUTPUT
		Y :	WORD;
	END_VAR

	VAR
		last :	UDINT;
		tx :	UDINT;
		init :	BOOL;
		tmp :	DINT;
		T_PLC_MS :	T_PLC_MS_Block;
	END_VAR

	T_PLC_MS();
	tx:= T_PLC_MS.T_PLC_MS;

	IF NOT init OR T = T#0s THEN
		init := TRUE;
		last := tx;
		Y := X;
	ELSIF Y = X THEN
		last := tx;
	ELSE
		tmp := UINT_TO_DINT(WORD_TO_UINT(X) - WORD_TO_UINT(Y)) * UDINT_TO_DINT(tx - last) / TIME_TO_DINT(T);
		IF tmp <> DINT#0 THEN
			Y := DINT_TO_WORD(WORD_TO_DINT(Y) + tmp);
			last := tx;
		END_IF;
	END_IF;

END_FUNCTION_BLOCK

PROGRAM program0
  VAR
	X :	WORD;
	T :	TIME;

	Y :	WORD;

	func_block : FILTER_W;
  END_VAR
	func_block.X  := X;
	func_block.T  := T;
	func_block();
	Y := func_block.Y;
END_PROGRAM

CONFIGURATION Config0
	VAR_GLOBAL
		PLC_TICKS_PER_SEC :	INT;
		PLC_SYS_TICK_CNT :	DINT;
	END_VAR
	RESOURCE Res0 ON PLC
		TASK task0(INTERVAL := T#20ms,PRIORITY := 0);
		PROGRAM instance0 WITH task0 : program0;
	END_RESOURCE
END_CONFIGURATION

(* ---- FILTER_WAV.ST ---- *)
TYPE
  oscat_arr_0_15              : ARRAY [0..15]   OF REAL;
END_TYPE

FUNCTION INC1:INT

	VAR_INPUT
		X :	INT;
		N :	INT;
	END_VAR

	IF X >= N - 1 THEN
		INC1 := 0;
	ELSE
		INC1 := X + 1;
	END_IF;
END_FUNCTION

FUNCTION DEC1:INT

	VAR_INPUT
		X :	INT;
		N :	INT;
	END_VAR

	IF X = 0 THEN
		DEC1 := N - 1;
	ELSE
		DEC1 := X - 1;
	END_IF;

END_FUNCTION

FUNCTION_BLOCK FILTER_WAV
	VAR_INPUT
		X :	REAL;
		W :	oscat_arr_0_15;
		RST :	BOOL;
	END_VAR

	VAR_OUTPUT
		Y :	REAL;
	END_VAR

	VAR
		init :	BOOL;
		buffer :	oscat_arr_0_15;
		i :	INT;
		n :	INT;
	END_VAR

	IF NOT init OR rst THEN
		init := TRUE;
		FOR i := 0 TO 15 DO
			buffer[i] := X;
		END_FOR;
		i := 15;
		Y := X;
	ELSE
		i := INC1(i, 16);
		buffer[i] := X;
	END_IF;

	Y := 0.0;
	FOR n := 0 TO 15 DO
		Y := buffer[i] * W[n] + Y;
		i := DEC1(i, 16);
	END_FOR;
END_FUNCTION_BLOCK

PROGRAM program0
  VAR
	X :	REAL;
	W :	oscat_arr_0_15;
	RST :	BOOL;

	Y :	REAL;

	func_block : FILTER_WAV;
  END_VAR
	func_block.X  := X;
	func_block.W  := W;
	func_block.RST  := RST;
	func_block();
	Y := func_block.Y;
END_PROGRAM

CONFIGURATION Config0

	RESOURCE Res0 ON PLC
		TASK task0(INTERVAL := T#20ms,PRIORITY := 0);
		PROGRAM instance0 WITH task0 : program0;
	END_RESOURCE
END_CONFIGURATION

(* ---- FINDB.ST ---- *)
FUNCTION_BLOCK FINDB_Block

	VAR_INPUT
		STR1 :	STRING;
		STR2 :	STRING;
	END_VAR

	VAR_OUTPUT
		FINDB :	INT;
	END_VAR

	VAR
		pos :	INT;
		length :	INT;
		string_temp :	STRING;
	END_VAR

	length := LEN(str2);
	pos := LEN(str1) - length +1;
	WHILE (pos >= 1) DO
		string_temp := MID(str1,length,pos);
		IF EQ_STRING(string_temp,str2) THEN
			FindB := pos;
			RETURN;
		END_IF;
	pos := pos -1;
	END_WHILE;
	FindB := 0;

END_FUNCTION_BLOCK

PROGRAM program0
  VAR
		STR1 :	STRING;
		STR2 :	STRING;

		FINDB :	INT;

	func_block : FINDB_Block;
  END_VAR
	func_block.STR1  := STR1;
	func_block.STR2  := STR2;
	func_block();
	FINDB := func_block.FINDB;
END_PROGRAM

CONFIGURATION Config0

	RESOURCE Res0 ON PLC
		TASK task0(INTERVAL := T#20ms,PRIORITY := 0);
		PROGRAM instance0 WITH task0 : program0;
	END_RESOURCE
END_CONFIGURATION

(* ---- FINDP.ST ---- *)
FUNCTION_BLOCK FINDP_Block

	VAR_INPUT
		STR :	STRING;
		SRC :	STRING;
		POS :	INT;
	END_VAR

	VAR_OUTPUT
		FINDP :	INT;
	END_VAR

	VAR
		i :	INT;
		ls :	INT;
		lx :	INT;
		stp :	INT;
		st_tmp :	STRING;
	END_VAR

	ls := LEN(str);
	lx := LEN(src);
	IF ls < lx OR lx = 0 THEN RETURN; END_IF;
	stp := ls - lx + 1;
	FOR i := MAX(pos,1) TO stp DO
		st_tmp := MID(str,lx,i);
		IF EQ_STRING(st_tmp,src) THEN
			FINDP := i;
			RETURN;
		END_IF;
	END_FOR;
	FINDP := 0;

END_FUNCTION_BLOCK

PROGRAM program0

	VAR
		STR :	STRING;
		SRC :	STRING;
		POS :	INT;

        FINDP :	INT;
		func_block : FINDP_Block;
	END_VAR
		func_block.STR := STR;
		func_block.SRC := SRC;
		func_block.POS := POS;
		func_block();
		FINDP := func_block.FINDP;

END_PROGRAM

CONFIGURATION Config0

	RESOURCE Res0 ON PLC
		TASK task0(INTERVAL := T#20ms,PRIORITY := 0);
		PROGRAM instance0 WITH task0 : program0;
	END_RESOURCE

END_CONFIGURATION

(* ---- FIX.ST ---- *)
FUNCTION _BYTE_TO_INT:INT
	VAR_INPUT
		IN :	BYTE;
	END_VAR

	_BYTE_TO_INT := USINT_TO_INT(BYTE_TO_USINT(IN));
END_FUNCTION

FUNCTION_BLOCK CHR_TO_STRING_Block
	VAR_INPUT
		C :	BYTE;
	END_VAR

	VAR_OUTPUT
		CHR_TO_STRING :	STRING;
	END_VAR

	CHR_TO_STRING := BYTE_TO_STRING(C);

END_FUNCTION_BLOCK

FUNCTION BIT_OF_DWORD : BOOL
  VAR_INPUT
    IN : DWORD;
    N : INT;
  END_VAR

  BIT_OF_DWORD := (SHR(in,N) AND 16#00000001) > 0;
  (* from OSCAT library; www.oscat.de  *)
END_FUNCTION

FUNCTION_BLOCK FILL_Block
	VAR_INPUT
		C :	BYTE;
		L :	INT;
	END_VAR

	VAR_OUTPUT
		FILL :	STRING;
	END_VAR

	VAR
		N :	BYTE;
		I :	INT;
		sx :	STRING;
		CHR_TO_STRING :	CHR_TO_STRING_Block;
		FILL_tmp :	STRING;
	END_VAR

	CHR_TO_STRING(C:=c);
	Sx:=CHR_TO_STRING.CHR_TO_STRING;
	(* create string *)
	N := INT_TO_BYTE(LIMIT(0,L,80));
	(* create a string of characters to be connected to str *)
	FILL := '';
	FOR i := 1 TO 8 DO
		FILL_tmp := FILL;
		FILL := CONCAT(FILL_tmp,FILL);
		IF BIT_OF_DWORD(BYTE_TO_DWORD(N),7) THEN FILL := CONCAT(FILL,Sx); END_IF;
		N := SHL(N,1);
	END_FOR;
END_FUNCTION_BLOCK

FUNCTION_BLOCK FIX_Block

	VAR_INPUT
		STR :	STRING;
		L :	INT;
		C :	BYTE;
		M :	INT;
	END_VAR

	VAR_OUTPUT
		FIX :	STRING;
	END_VAR

	VAR
		N :	INT;
		FILL :	FILL_Block;
	END_VAR

	N := LIMIT(0,L,255) - LEN(str);
	IF N <= 0 THEN
		(* truncate the string at length N *)
		IF M = 1 THEN
			FIX := RIGHT(str,L);
		ELSE
			FIX := LEFT(str,L);
		END_IF;
	ELSIF M = 1 THEN
		(* connect fill characters at the beginning *)
		FILL(C:=C,L:=N);
		FIX := CONCAT(FILL.FILL,str);
	ELSIF M = 2 THEN
		(* center str beween fill characters *)
		(* for an uneven number of fill characters, there is one more at the end *)
		FILL(C:=C,L:=_BYTE_TO_INT(SHR(INT_TO_BYTE(N+1),1)));
		FIX := CONCAT(str,FILL.FILL);
		FILL(C:=C,L:=_BYTE_TO_INT(SHR(INT_TO_BYTE(N),1)));
		FIX := CONCAT(FILL.FILL,FIX);
	ELSE
		(* connect fill characters at the end *)
		FILL(C:=C,L:=N);
		FIX := CONCAT(str,FILL.FILL);
	END_IF;

END_FUNCTION_BLOCK

PROGRAM program0
  VAR
	STR :	STRING;
	L   :	INT;
	C   :	BYTE;
	M   :	INT;

	FIX :	STRING;

	func_block : FIX_Block;
  END_VAR
	func_block.STR:=STR;
	func_block.L  :=L  ;
	func_block.C  :=C  ;
	func_block.M  :=M  ;
	func_block();
	FIX := func_block.FIX;
END_PROGRAM

CONFIGURATION Config0
  RESOURCE Res0 ON PLC
    TASK task0(INTERVAL := T#20ms,PRIORITY := 0);
    PROGRAM instance0 WITH task0 : program0;
  END_RESOURCE
END_CONFIGURATION

(* ---- FLOW_CONTROL.ST ---- *)
FUNCTION UDINT_TO_TIME2:TIME

	VAR_INPUT
		IN :	UDINT;
	END_VAR

	UDINT_TO_TIME2 := DINT_TO_TIME(UDINT_TO_DINT(IN));

END_FUNCTION

FUNCTION_BLOCK T_PLC_MS_block
	VAR_OUTPUT
		T_PLC_MS :	UDINT;
	END_VAR

	VAR_EXTERNAL
		PLC_TICKS_PER_SEC :	INT;
		PLC_SYS_TICK_CNT :	DINT;
	END_VAR

	VAR
		debug :	BOOL;(*Debug-Mode ON / OFF*)
		N :	INT;(*Debug-Faktor*)
		Offset :	UDINT;(*Debug-Offset*)
		temp :	DWORD := DWORD#1;(*Debug-Offset*)
		mode :	BOOL;(*modus*)
		faktor :	UDINT;(*Systemtakt-Faktor*)
		init :	BOOL;
		v_plc_ticks_per_sec :	UDINT;
		base :	UDINT := UDINT#1000;
	END_VAR

	IF init = FALSE THEN
		v_plc_ticks_per_sec := INT_TO_UDINT(PLC_TICKS_PER_SEC);
		IF v_plc_ticks_per_sec = UDINT#1024 THEN
			faktor := UDINT#1;
			mode := FALSE;
		ELSIF v_plc_ticks_per_sec > UDINT#0 THEN
			IF v_plc_ticks_per_sec <= base THEN
				faktor := base / v_plc_ticks_per_sec;
				mode := FALSE;
			ELSE
				faktor := v_plc_ticks_per_sec / base;
				mode := TRUE;
			END_IF;
		ELSE
			faktor := UDINT#1;
		END_IF;
		init := TRUE;
	END_IF;

	IF mode THEN
		T_PLC_MS := DINT_TO_UDINT(PLC_SYS_TICK_CNT) / faktor;
	ELSE
		T_PLC_MS := DINT_TO_UDINT(PLC_SYS_TICK_CNT) * faktor;
	END_IF;

	IF debug THEN
		T_PLC_MS := (DWORD_TO_UDINT(SHL(UDINT_TO_DWORD(T_PLC_MS),N) OR SHL(temp,N)) - UDINT#1) + Offset;
	END_IF;
END_FUNCTION_BLOCK

FUNCTION_BLOCK TP_1D
	VAR_INPUT
		IN :	BOOL;
		PT1 :	TIME;
		PTD :	TIME;
		RST :	BOOL;
	END_VAR

	VAR_OUTPUT
		Q :	BOOL;
		W :	BOOL;
	END_VAR

	VAR
		tx :	TIME;
		start :	TIME;
		ix :	BOOL;
		T_PLC_MS :	T_PLC_MS_block;
	END_VAR

	T_PLC_MS();
	tx := UDINT_TO_TIME(T_PLC_MS.T_PLC_MS);

	IF RST THEN
		Q := FALSE;
		rst := FALSE;
		W := FALSE;
	ELSIF W THEN
		IF tx - start >= PTD THEN
			W := FALSE;
		END_IF;
	ELSIF IN AND NOT ix THEN
		Q := TRUE;
		start := tx;
		in := FALSE;
	ELSIF tx - start >= PT1 THEN
		Q := FALSE;
		W := TRUE;
		start := tx;
	END_IF;

	ix := IN;

END_FUNCTION_BLOCK

FUNCTION_BLOCK FLOW_CONTROL
	VAR_INPUT
		IN :	BOOL;
		REQ :	BOOL;
		ENQ :	BOOL;
		RST :	BOOL := FALSE;
		T_AUTO :	TIME := T#1h;
		T_DELAY :	TIME := T#23h;
	END_VAR

	VAR_OUTPUT
		Q :	BOOL;
		STATUS :	BYTE;
	END_VAR

	VAR
		timer :	TP_1D;
	END_VAR

	STATUS := BYTE#100;
	IF RST THEN
		Q := FALSE;
		timer(rst := TRUE);
		timer.RST := FALSE;
		STATUS := BYTE#103;
	ELSIF ENQ THEN
		IF IN THEN
			status := BYTE#101;
		END_IF;
		IF REQ THEN
			(* timer will generate a timed pulse after TP goes high *)
			timer.PT1 := T_AUTO;
			timer.PTD := T_DELAY;
			timer.IN := TRUE;
			STATUS := BYTE#102;
		END_IF;
	END_IF;

	timer();
	timer.IN := FALSE;
	Q := (IN AND ENQ) OR timer.Q;
END_FUNCTION_BLOCK

PROGRAM program0
  VAR
	IN      :	BOOL;
	REQ     :	BOOL;
	ENQ     :	BOOL;
	RST     :	BOOL ;
	T_AUTO  :	TIME ;
	T_DELAY :	TIME ;

	Q      :	BOOL;
	STATUS :	BYTE;

	func_block : FLOW_CONTROL;
  END_VAR
	func_block.IN     :=IN     ;
	func_block.REQ    :=REQ    ;
	func_block.ENQ    :=ENQ    ;
	func_block.RST    :=RST    ;
	func_block.T_AUTO :=T_AUTO ;
	func_block.T_DELAY:=T_DELAY;
	func_block();
	Q     := func_block.Q     ;
	STATUS:= func_block.STATUS;
END_PROGRAM

CONFIGURATION Config0
	VAR_GLOBAL
		PLC_TICKS_PER_SEC :	INT;
		PLC_SYS_TICK_CNT :	DINT;
	END_VAR
	RESOURCE Res0 ON PLC
		TASK task0(INTERVAL := T#20ms,PRIORITY := 0);
		PROGRAM instance0 WITH task0 : program0;
	END_RESOURCE
END_CONFIGURATION

(* ---- FLOW_CONTROL_4.ST ---- *)
FUNCTION_BLOCK FLOW_CONTROL_4
	VAR_INPUT
		I0 :	BOOL;
		I1 :	BOOL;
		I2 :	BOOL;
		I3 :	BOOL;
		PR :	BOOL;
		ICE :	BOOL;
		DIAG :	BOOL;
		ENQ :	BOOL;
		RST :	BOOL := FALSE;
		TD_WAIT :	TIME := T#5s;
		TD_S :	TIME := T#10s;
		TD_0 :	TIME := T#10s;
	END_VAR

	VAR_OUTPUT
		QS :	BOOL;
		Q0 :	BOOL;
		Q1 :	BOOL;
		Q2 :	BOOL;
		Q3 :	BOOL;
		ERROR :	BOOL;
		STATUS :	BYTE;
	END_VAR

	VAR
		state :	INT;
		timer :	TP;
	END_VAR

	IF RST THEN
		STATUS := BYTE#100;
		state := 0;
		error := FALSE;

	ELSIF DIAG THEN
		CASE state OF
			0 : (* start diag operation *)
				(* close all valves and pressurize the system *)
				QS := TRUE;
				Q0 := FALSE;
				Q1 := FALSE;
				Q2 := FALSE;
				Q3 := FALSE;
				timer(in := TRUE, pt := TD_WAIT);
				timer.IN := FALSE;
				state := 1;
			1 : (* wait for TD_wait *)
				timer();
				IF NOT timer.Q THEN
					QS := FALSE;
					timer(in := TRUE, pt := TD_S);
					timer.IN := FALSE;
					state := 2;
				END_IF;
			2:	(* wait for safety valve pressure test *)
				timer();
				IF NOT timer.Q THEN
					IF NOT pr THEN
						(* system pressure failure *)
						ERROR := TRUE;
						STATUS := BYTE#1;
						RETURN;
					END_IF;
					timer(in := TRUE, pt := TD_0);
					timer.IN := FALSE;
					Q0 := TRUE;
					state := 3;
				END_IF;
			3:	(* wait for pressure on Q0 to hold TD_0 *)
				timer();
				IF NOT timer.Q THEN
					IF NOT pr THEN
						(* valve 0 pressure failure *)
						ERROR := TRUE;
						STATUS := BYTE#1;
						RETURN;
					END_IF;
					Q0 := FALSE;
					QS := TRUE;
				END_IF;
		END_CASE;
	ELSIF ICE THEN
		(* when frost is present we close the safety valve and open all other valves to depressurize the valves *)
		QS := FALSE;
		Q0 := TRUE;
		Q1 := TRUE;
		Q2 := TRUE;
		Q3 := TRUE;
		STATUS := BYTE#110;

	ELSIF NOT error AND ENQ THEN
			Q0 := I0;
			Q1 := I1;
			Q2 := I2;
			Q3 := I3;
			QS := Q0 OR Q1 OR Q2 OR Q3;
			STATUS := BYTE#100;

			(* maximum ontime check *)
	ELSE
		Q0 := FALSE;
		Q1 := FALSE;
		Q2 := FALSE;
		Q3 := FALSE;
	END_IF;

END_FUNCTION_BLOCK

PROGRAM program0
  VAR
		I0   :	BOOL;
		I1   :	BOOL;
		I2   :	BOOL;
		I3   :	BOOL;
		PR   :	BOOL;
		ICE  :	BOOL;
		DIAG :	BOOL;
		ENQ  :	BOOL;
		RST  :	BOOL ;
		TD_WAIT :	TIME;
		TD_S    :	TIME;
		TD_0    :	TIME;

		QS     :	BOOL;
		Q0     :	BOOL;
		Q1     :	BOOL;
		Q2     :	BOOL;
		Q3     :	BOOL;
		ERROR  :	BOOL;
		STATUS :	BYTE;

	func_block : FLOW_CONTROL_4;
  END_VAR
	func_block.I0  :=I0  ;
	func_block.I1  :=I1  ;
	func_block.I2  :=I2  ;
	func_block.I3  :=I3  ;
	func_block.PR  :=PR  ;
	func_block.ICE :=ICE ;
	func_block.DIAG:=DIAG;
	func_block.ENQ :=ENQ ;
	func_block.RST :=RST ;
	func_block.TD_WAIT:=TD_WAIT;
	func_block.TD_S   :=TD_S   ;
	func_block.TD_0   :=TD_0   ;
	func_block();
	QS    := func_block.QS    ;
	Q0    := func_block.Q0    ;
	Q1    := func_block.Q1    ;
	Q2    := func_block.Q2    ;
	Q3    := func_block.Q3    ;
	ERROR := func_block.ERROR ;
	STATUS:= func_block.STATUS;

END_PROGRAM

CONFIGURATION Config0
  RESOURCE Res0 ON PLC
    TASK task0(INTERVAL := T#20ms,PRIORITY := 0);
    PROGRAM instance0 WITH task0 : program0;
  END_RESOURCE
END_CONFIGURATION

(* ---- FLOW_METER.ST ---- *)
FUNCTION_BLOCK T_PLC_MS_block
	VAR_OUTPUT
		T_PLC_MS :	UDINT;
	END_VAR

	VAR_EXTERNAL
		PLC_TICKS_PER_SEC :	INT;
		PLC_SYS_TICK_CNT :	DINT;
	END_VAR

	VAR
		debug :	BOOL;(*Debug-Mode ON / OFF*)
		N :	INT;(*Debug-Faktor*)
		Offset :	UDINT;(*Debug-Offset*)
		temp :	DWORD := DWORD#1;(*Debug-Offset*)
		mode :	BOOL;(*modus*)
		faktor :	UDINT;(*Systemtakt-Faktor*)
		init :	BOOL;
		v_plc_ticks_per_sec :	UDINT;
		base :	UDINT := UDINT#1000;
	END_VAR

	IF init = FALSE THEN
		v_plc_ticks_per_sec := INT_TO_UDINT(PLC_TICKS_PER_SEC);
		IF v_plc_ticks_per_sec = UDINT#1024 THEN
			faktor := UDINT#1;
			mode := FALSE;
		ELSIF v_plc_ticks_per_sec > UDINT#0 THEN
			IF v_plc_ticks_per_sec <= base THEN
				faktor := base / v_plc_ticks_per_sec;
				mode := FALSE;
			ELSE
				faktor := v_plc_ticks_per_sec / base;
				mode := TRUE;
			END_IF;
		ELSE
			faktor := UDINT#1;
		END_IF;
		init := TRUE;
	END_IF;

	IF mode THEN
		T_PLC_MS := DINT_TO_UDINT(PLC_SYS_TICK_CNT) / faktor;
	ELSE
		T_PLC_MS := DINT_TO_UDINT(PLC_SYS_TICK_CNT) * faktor;
	END_IF;

	IF debug THEN
		T_PLC_MS := (DWORD_TO_UDINT(SHL(UDINT_TO_DWORD(T_PLC_MS),N) OR SHL(temp,N)) - UDINT#1) + Offset;
	END_IF;
END_FUNCTION_BLOCK

FUNCTION_BLOCK INTEGRATE

	VAR_INPUT
		E :	BOOL := TRUE;
		X :	REAL;
		K :	REAL := 1.0;
	END_VAR

	VAR_IN_OUT
		Y :	REAL;
	END_VAR

	VAR
		X_last :	REAL;
		init :	BOOL;
		T_PLC_MS :	T_PLC_MS_block;
		last :	UDINT;
		tx :	UDINT;
	END_VAR

	T_PLC_MS();
	tx:= T_PLC_MS.T_PLC_MS;

	IF NOT init THEN
		init := TRUE;
		X_last := X;
	ELSIF E THEN
		Y := (X + X_LAST) * 0.5E-3 * UDINT_TO_REAL(tx-last) * K + Y;
		X_last := X;
	END_IF;
	last := tx;

END_FUNCTION_BLOCK

FUNCTION _INT_TO_UDINT:UDINT
	VAR_INPUT
		IN :	INT;
	END_VAR

	_INT_TO_UDINT := DINT_TO_UDINT(INT_TO_DINT(IN));
END_FUNCTION

FUNCTION FLOOR : INT
	VAR_INPUT
		x : REAL;
	END_VAR

	FLOOR := REAL_TO_INT(X);
	IF INT_TO_REAL(FLOOR) > X THEN
		floor := floor - 1;
	END_IF;
END_FUNCTION

FUNCTION_BLOCK FLOW_METER
	VAR_INPUT
		VX :	REAL;
		E :	BOOL;
		RST :	BOOL;
		PULSE_MODE :	BOOL;
		UPDATE_TIME :	TIME := T#1s;
	END_VAR

	VAR_OUTPUT
		F :	REAL;
	END_VAR

	VAR_IN_OUT
		X :	REAL;
		Y :	UDINT;
	END_VAR

	VAR
		T_PLC_MS :	T_PLC_MS_block;
		tx :	TIME;
		tl :	TIME;
		int1 :	INTEGRATE;
		init :	BOOL;
		e_last :	BOOL;
		tmp :	INT;
		x_last :	REAL;
		y_last :	UDINT;
	END_VAR

	IF NOT init THEN	(* init on power up *)
		init := TRUE;
		tl := tx;
		x_last := X;
		y_last := Y;
		int1.K := 2.7777777777777777E-4;
	END_IF;

	int1(E := NOT (RST OR PULSE_MODE) AND E, X := VX, Y := X);	(* gated operation *)
	X := int1.Y;

	IF RST THEN		(* reset *)
		X := 0.0;
		Y := UDINT#0;
		tl := tx;
		x_last := 0.0;
		y_last := UDINT#0;
	ELSIF E AND PULSE_MODE THEN	(* check for pulse mode *)
		IF NOT e_last THEN X := X + VX; END_IF;
	END_IF;
	e_last := E;

	(* reduce X to be less than 1 and increase Y respectively *)
	IF X > 1.0 THEN
		tmp := FLOOR(X);
		Y := Y + _INT_TO_UDINT(tmp);
		X := X - INT_TO_REAL(tmp);
	END_IF;

	(* calculate the current flow *)
	T_PLC_MS();
	tx := UDINT_TO_TIME(T_PLC_MS.T_PLC_MS);
	IF tx - tl >= UPDATE_TIME AND UPDATE_TIME > t#0s THEN
		F := (UDINT_TO_REAL(Y - y_last) + X - x_last) / TIME_TO_REAL(tx - tl) * 3.6E6;
		y_last := Y;
		x_last := X;
		tl := tx;
	END_IF;

END_FUNCTION_BLOCK

PROGRAM program0
  VAR
	VX :	REAL;
	E :	BOOL;
	RST :	BOOL;
	PULSE_MODE :	BOOL;
	UPDATE_TIME :	TIME := T#1s;

	F :	REAL;

	X :	REAL;
	Y :	UDINT;

	func_block : FLOW_METER;
  END_VAR
	func_block.VX:=VX;
	func_block.E:=E;
	func_block.RST:=RST;
	func_block.PULSE_MODE:=PULSE_MODE;
	func_block.UPDATE_TIME :=UPDATE_TIME ;
	func_block.X:=X;
	func_block.Y:=Y;
	func_block();
	F:= func_block.F;
	X:= func_block.X;
	Y:= func_block.Y;
END_PROGRAM

CONFIGURATION Config0
	VAR_GLOBAL
		PLC_TICKS_PER_SEC :	INT;
		PLC_SYS_TICK_CNT :	DINT;
	END_VAR
	RESOURCE Res0 ON PLC
		TASK task0(INTERVAL := T#20ms,PRIORITY := 0);
		PROGRAM instance0 WITH task0 : program0;
	END_RESOURCE
END_CONFIGURATION

(* ---- FT_AVG.ST ---- *)
TYPE
	oscat_delay_buf             : ARRAY [0..31]   OF REAL;
END_TYPE

FUNCTION INC1:INT

	VAR_INPUT
		X :	INT;
		N :	INT;
	END_VAR

	IF X >= N - 1 THEN
		INC1 := 0;
	ELSE
		INC1 := X + 1;
	END_IF;
END_FUNCTION

FUNCTION_BLOCK DELAY

	VAR_INPUT
		IN :	REAL;
		N :	INT;
		RST :	BOOL;
	END_VAR

	VAR_OUTPUT
		OUT :	REAL;
	END_VAR

	VAR
		buf :	oscat_delay_buf;
		i :	INT;
		init :	BOOL;
		stop :	INT;
	END_VAR

	stop := LIMIT(0,N,32) - 1;
	IF rst OR NOT init THEN
		init := TRUE;
		FOR i := 0 TO stop DO buf[i] := in; END_FOR;
		out := in;
		i := 0;
	ELSIF stop < 0 THEN
		out := in;
	ELSE
		out := buf[i];
		buf[i] := in;
		i := INC1(i, N);
	END_IF;

END_FUNCTION_BLOCK

FUNCTION_BLOCK FT_AVG

	VAR_INPUT
		IN :	REAL;
		E :	BOOL := TRUE;
		N :	INT := INT#32;
		RST :	BOOL;
	END_VAR

	VAR_OUTPUT
		AVG :	REAL;
	END_VAR

	VAR
		buff :	delay;
		i :	INT;
		init :	BOOL;
	END_VAR

	buff.N := LIMIT(0, N, 32);

	IF NOT init OR rst THEN
		FOR i := 1 TO N DO
			buff(in := in);
		END_FOR;
		avg := in;
		init := TRUE;
	ELSIF E THEN
		buff(in := in);
		avg := avg + (in - buff.out ) / INT_TO_REAL(N);
	END_IF;

END_FUNCTION_BLOCK

PROGRAM program0
  VAR
		IN  :	REAL;
		E   :	BOOL;
		N   :	INT;
		RST :	BOOL;

		AVG :	REAL;

	func_block : FT_AVG;
  END_VAR
	func_block.IN :=IN ;
	func_block.E  :=E  ;
	func_block.N  :=N  ;
	func_block.RST:=RST;
	func_block();
	AVG := func_block.AVG;
END_PROGRAM

CONFIGURATION Config0
  RESOURCE Res0 ON PLC
    TASK task0(INTERVAL := T#20ms,PRIORITY := 0);
    PROGRAM instance0 WITH task0 : program0;
  END_RESOURCE
END_CONFIGURATION
